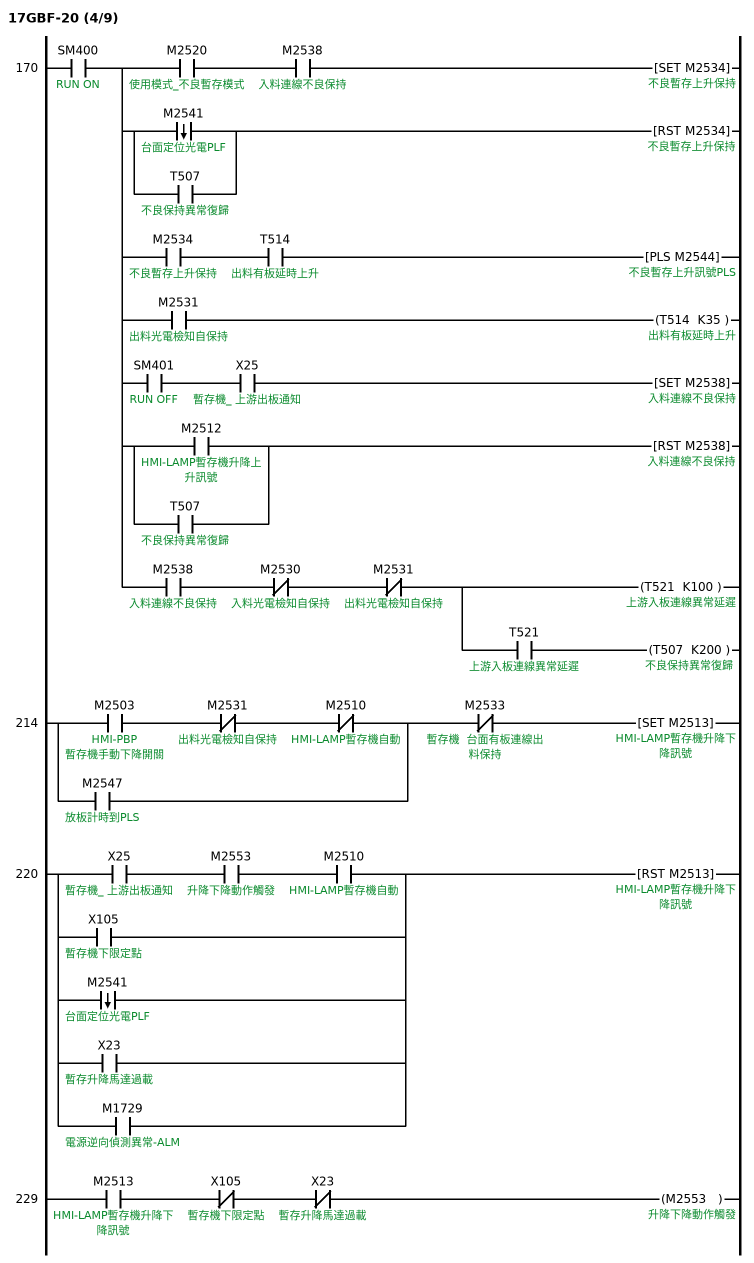
[picture p144: ladder of 17GBF-20, rungs at steps 170 to 229]
170   LD      SM400  ; RUN ON
      MPS
      AND     M2520  ; 使用模式_不良暫存模式
      AND     M2538  ; 入料連線不良保持
      SET     M2534  ; 不良暫存上升保持
      MRD
      LDF     M2541  ; 台面定位光電PLF
      OR      T507  ; 不良保持異常復歸
      ANB
      RST     M2534  ; 不良暫存上升保持
      MRD
      AND     M2534  ; 不良暫存上升保持
      AND     T514  ; 出料有板延時上升
      PLS     M2544  ; 不良暫存上升訊號PLS
      MRD
      AND     M2531  ; 出料光電檢知自保持
      OUT     T514 K35  ; 出料有板延時上升
      MRD
      AND     SM401  ; RUN OFF
      AND     X25  ; 暫存機_ 上游出板通知
      SET     M2538  ; 入料連線不良保持
      MRD
      LD      M2512  ; HMI-LAMP暫存機升降上升訊號
      OR      T507  ; 不良保持異常復歸
      ANB
      RST     M2538  ; 入料連線不良保持
      MPP
      AND     M2538  ; 入料連線不良保持
      ANI     M2530  ; 入料光電檢知自保持
      ANI     M2531  ; 出料光電檢知自保持
      OUT     T521 K100  ; 上游入板連線異常延遲
      AND     T521  ; 上游入板連線異常延遲
      OUT     T507 K200  ; 不良保持異常復歸
214   LD      M2503  ; HMI-PBP 暫存機手動下降開關
      ANI     M2531  ; 出料光電檢知自保持
      ANI     M2510  ; HMI-LAMP暫存機自動
      OR      M2547  ; 放板計時到PLS
      ANI     M2533  ; 暫存機  台面有板連線出料保持
      SET     M2513  ; HMI-LAMP暫存機升降下降訊號
220   LD      X25  ; 暫存機_ 上游出板通知
      AND     M2553  ; 升降下降動作觸發
      AND     M2510  ; HMI-LAMP暫存機自動
      OR      X105  ; 暫存機下限定點
      ORF     M2541  ; 台面定位光電PLF
      OR      X23  ; 暫存升降馬達過載
      OR      M1729  ; 電源逆向偵測異常-ALM
      RST     M2513  ; HMI-LAMP暫存機升降下降訊號
229   LD      M2513  ; HMI-LAMP暫存機升降下降訊號
      ANI     X105  ; 暫存機下限定點
      ANI     X23  ; 暫存升降馬達過載
      OUT     M2553  ; 升降下降動作觸發
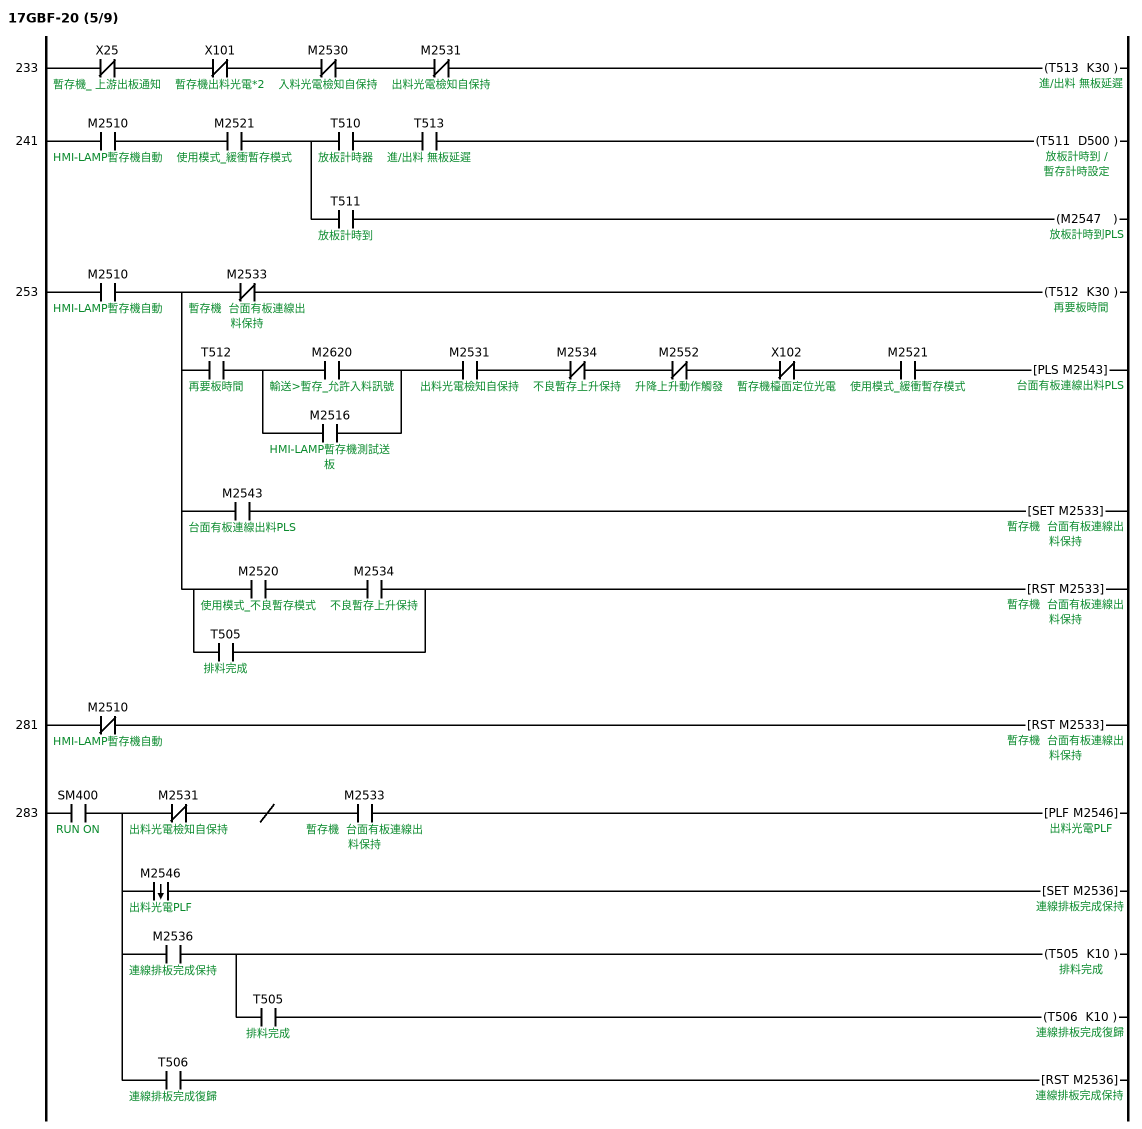
233   LDI     X25  ; 暫存機_ 上游出板通知
      ANI     X101  ; 暫存機出料光電*2
      ANI     M2530  ; 入料光電檢知自保持
      ANI     M2531  ; 出料光電檢知自保持
      OUT     T513 K30  ; 進/出料 無板延遲
241   LD      M2510  ; HMI-LAMP暫存機自動
      AND     M2521  ; 使用模式_緩衝暫存模式
      MPS
      AND     T510  ; 放板計時器
      AND     T513  ; 進/出料 無板延遲
      OUT     T511 D500  ; 放板計時到 / 暫存計時設定
      MPP
      AND     T511  ; 放板計時到
      OUT     M2547  ; 放板計時到PLS
253   LD      M2510  ; HMI-LAMP暫存機自動
      MPS
      ANI     M2533  ; 暫存機  台面有板連線出料保持
      OUT     T512 K30  ; 再要板時間
      MRD
      AND     T512  ; 再要板時間
      LD      M2620  ; 輸送>暫存_允許入料訊號
      OR      M2516  ; HMI-LAMP暫存機測試送板
      ANB
      AND     M2531  ; 出料光電檢知自保持
      ANI     M2534  ; 不良暫存上升保持
      ANI     M2552  ; 升降上升動作觸發
      ANI     X102  ; 暫存機檯面定位光電
      AND     M2521  ; 使用模式_緩衝暫存模式
      PLS     M2543  ; 台面有板連線出料PLS
      MRD
      AND     M2543  ; 台面有板連線出料PLS
      SET     M2533  ; 暫存機  台面有板連線出料保持
      MPP
      LD      M2520  ; 使用模式_不良暫存模式
      AND     M2534  ; 不良暫存上升保持
      OR      T505  ; 排料完成
      ANB
      RST     M2533  ; 暫存機  台面有板連線出料保持
281   LDI     M2510  ; HMI-LAMP暫存機自動
      RST     M2533  ; 暫存機  台面有板連線出料保持
283   LD      SM400  ; RUN ON
      MPS
      ANI     M2531  ; 出料光電檢知自保持
      INV
      AND     M2533  ; 暫存機  台面有板連線出料保持
      PLF     M2546  ; 出料光電PLF
      MRD
      ANDF    M2546  ; 出料光電PLF
      SET     M2536  ; 連線排板完成保持
      MRD
      AND     M2536  ; 連線排板完成保持
      OUT     T505 K10  ; 排料完成
      AND     T505  ; 排料完成
      OUT     T506 K10  ; 連線排板完成復歸
      MPP
      AND     T506  ; 連線排板完成復歸
      RST     M2536  ; 連線排板完成保持
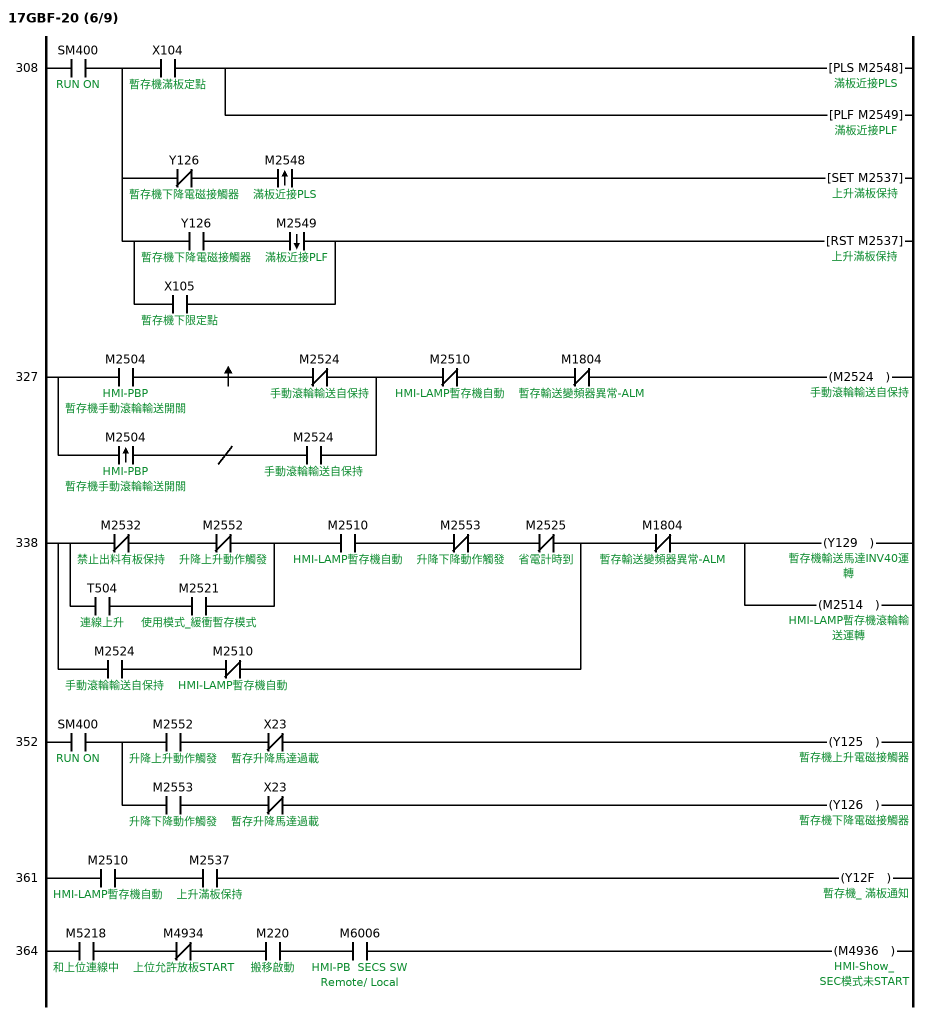
308   LD      SM400  ; RUN ON
      MPS
      AND     X104  ; 暫存機滿板定點
      PLS     M2548  ; 滿板近接PLS
      PLF     M2549  ; 滿板近接PLF
      MRD
      ANI     Y126  ; 暫存機下降電磁接觸器
      ANDP    M2548  ; 滿板近接PLS
      SET     M2537  ; 上升滿板保持
      MPP
      LD      Y126  ; 暫存機下降電磁接觸器
      ANDF    M2549  ; 滿板近接PLF
      OR      X105  ; 暫存機下限定點
      ANB
      RST     M2537  ; 上升滿板保持
327   LD      M2504  ; HMI-PBP 暫存機手動滾輪輸送開關
      MEP
      ANI     M2524  ; 手動滾輪輸送自保持
      LDP     M2504  ; HMI-PBP 暫存機手動滾輪輸送開關
      INV
      AND     M2524  ; 手動滾輪輸送自保持
      ORB
      ANI     M2510  ; HMI-LAMP暫存機自動
      ANI     M1804  ; 暫存輸送變頻器異常-ALM
      OUT     M2524  ; 手動滾輪輸送自保持
338   LDI     M2532  ; 禁止出料有板保持
      ANI     M2552  ; 升降上升動作觸發
      LD      T504  ; 連線上升
      AND     M2521  ; 使用模式_緩衝暫存模式
      ORB
      AND     M2510  ; HMI-LAMP暫存機自動
      ANI     M2553  ; 升降下降動作觸發
      ANI     M2525  ; 省電計時到
      LD      M2524  ; 手動滾輪輸送自保持
      ANI     M2510  ; HMI-LAMP暫存機自動
      ORB
      ANI     M1804  ; 暫存輸送變頻器異常-ALM
      OUT     Y129  ; 暫存機輸送馬達INV40運轉
      OUT     M2514  ; HMI-LAMP暫存機滾輪輸送運轉
352   LD      SM400  ; RUN ON
      MPS
      AND     M2552  ; 升降上升動作觸發
      ANI     X23  ; 暫存升降馬達過載
      OUT     Y125  ; 暫存機上升電磁接觸器
      MPP
      AND     M2553  ; 升降下降動作觸發
      ANI     X23  ; 暫存升降馬達過載
      OUT     Y126  ; 暫存機下降電磁接觸器
361   LD      M2510  ; HMI-LAMP暫存機自動
      AND     M2537  ; 上升滿板保持
      OUT     Y12F  ; 暫存機_ 滿板通知
364   LD      M5218  ; 和上位連線中
      ANI     M4934  ; 上位允許放板START
      AND     M220  ; 搬移啟動
      AND     M6006  ; HMI-PB  SECS SW  Remote/ Local
      OUT     M4936  ; HMI-Show_SEC模式未START
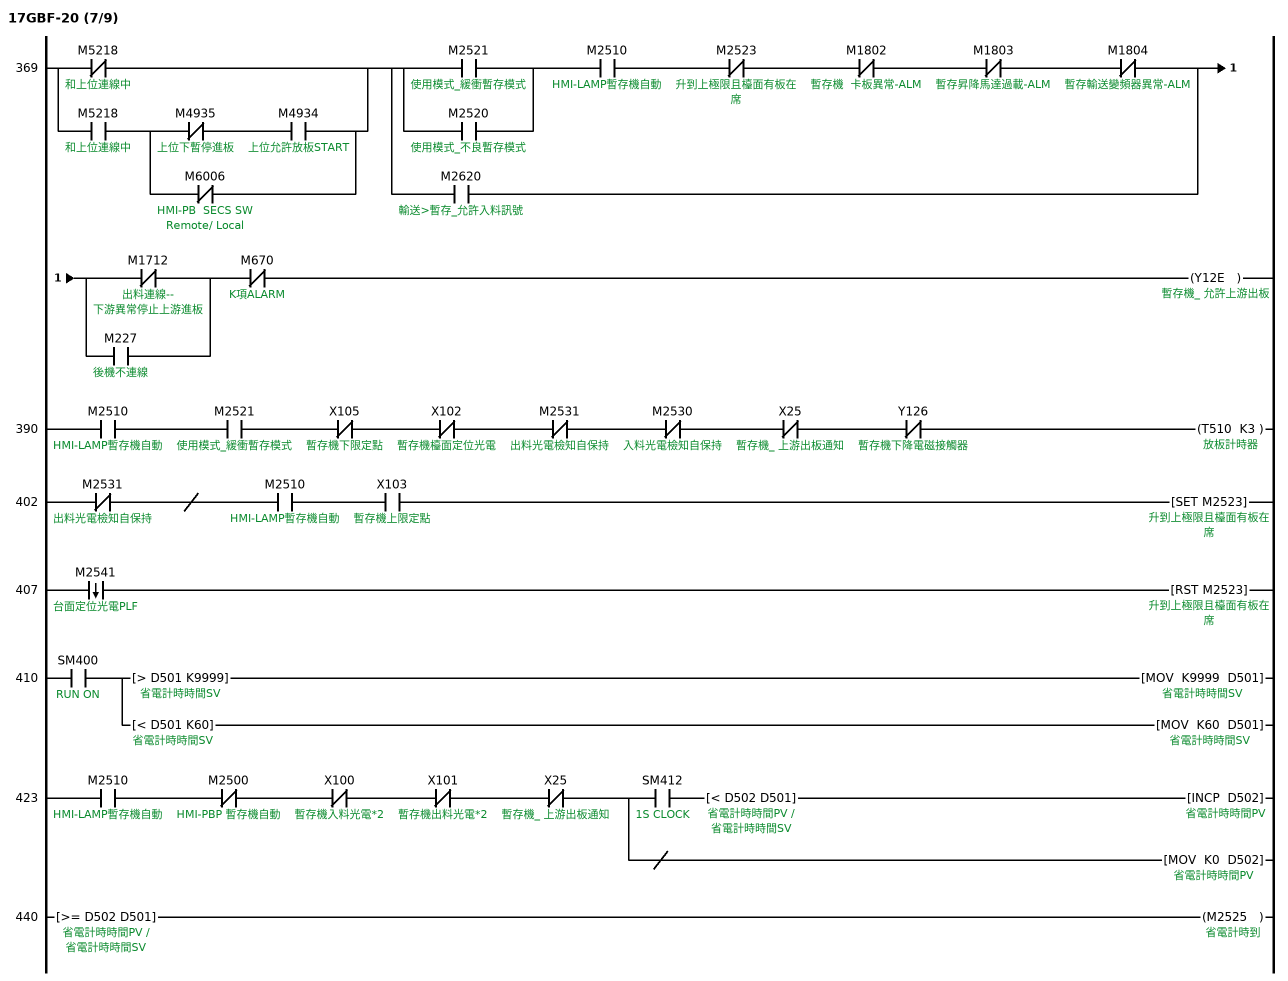
369   LDI     M5218  ; 和上位連線中
      LD      M5218  ; 和上位連線中
      LDI     M4935  ; 上位下暫停進板
      AND     M4934  ; 上位允許放板START
      ORI     M6006  ; HMI-PB  SECS SW  Remote/ Local
      ANB
      ORB
      LD      M2521  ; 使用模式_緩衝暫存模式
      OR      M2520  ; 使用模式_不良暫存模式
      AND     M2510  ; HMI-LAMP暫存機自動
      ANI     M2523  ; 升到上極限且檯面有板在席
      ANI     M1802  ; 暫存機  卡板異常-ALM
      ANI     M1803  ; 暫存昇降馬達過載-ALM
      ANI     M1804  ; 暫存輸送變頻器異常-ALM
      OR      M2620  ; 輸送>暫存_允許入料訊號
      ANB
      LDI     M1712  ; 出料連線--下游異常停止上游進板
      OR      M227  ; 後機不連線
      ANB
      ANI     M670  ; K項ALARM
      OUT     Y12E  ; 暫存機_ 允許上游出板
390   LD      M2510  ; HMI-LAMP暫存機自動
      AND     M2521  ; 使用模式_緩衝暫存模式
      ANI     X105  ; 暫存機下限定點
      ANI     X102  ; 暫存機檯面定位光電
      ANI     M2531  ; 出料光電檢知自保持
      ANI     M2530  ; 入料光電檢知自保持
      ANI     X25  ; 暫存機_ 上游出板通知
      ANI     Y126  ; 暫存機下降電磁接觸器
      OUT     T510 K3  ; 放板計時器
402   LDI     M2531  ; 出料光電檢知自保持
      INV
      AND     M2510  ; HMI-LAMP暫存機自動
      AND     X103  ; 暫存機上限定點
      SET     M2523  ; 升到上極限且檯面有板在席
407   LDF     M2541  ; 台面定位光電PLF
      RST     M2523  ; 升到上極限且檯面有板在席
410   LD      SM400  ; RUN ON
      MPS
      AND>    D501 K9999  ; 省電計時時間SV
      MOV     K9999 D501
      MPP
      AND<    D501 K60  ; 省電計時時間SV
      MOV     K60 D501
423   LD      M2510  ; HMI-LAMP暫存機自動
      ANI     M2500  ; HMI-PBP 暫存機自動
      ANI     X100  ; 暫存機入料光電*2
      ANI     X101  ; 暫存機出料光電*2
      ANI     X25  ; 暫存機_ 上游出板通知
      MPS
      AND     SM412  ; 1S CLOCK
      AND<    D502 D501  ; 省電計時時間PV / 省電計時時間SV
      INCP    D502
      MPP
      INV
      MOV     K0 D502
440   LD>=    D502 D501  ; 省電計時時間PV / 省電計時時間SV
      OUT     M2525  ; 省電計時到
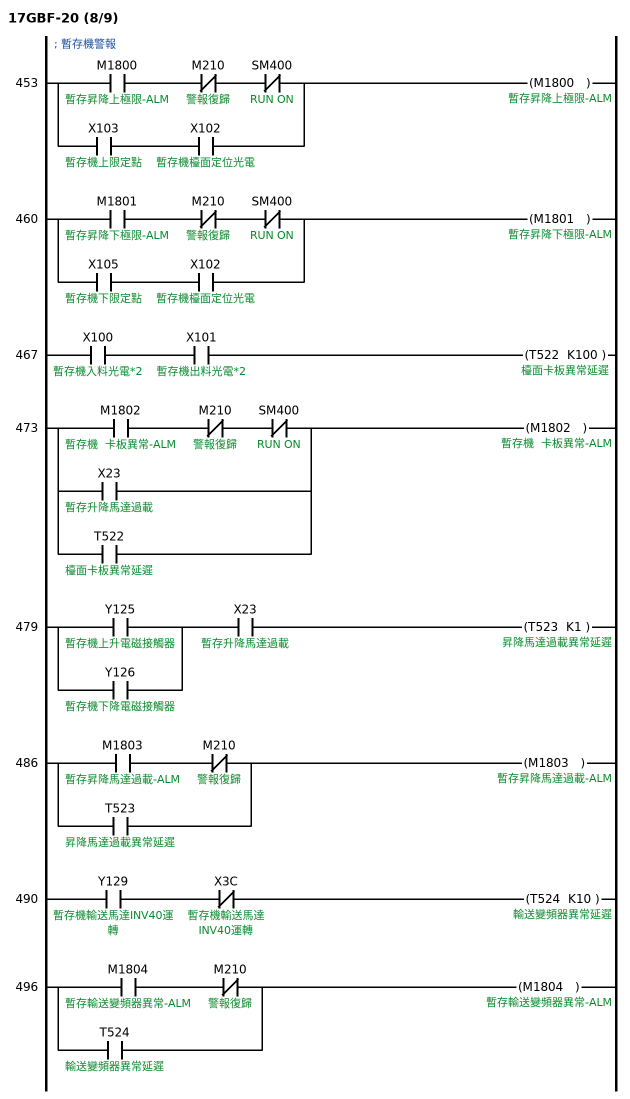
; 暫存機警報
453   LD      M1800  ; 暫存昇降上極限-ALM
      ANI     M210  ; 警報復歸
      ANI     SM400  ; RUN ON
      LD      X103  ; 暫存機上限定點
      AND     X102  ; 暫存機檯面定位光電
      ORB
      OUT     M1800  ; 暫存昇降上極限-ALM
460   LD      M1801  ; 暫存昇降下極限-ALM
      ANI     M210  ; 警報復歸
      ANI     SM400  ; RUN ON
      LD      X105  ; 暫存機下限定點
      AND     X102  ; 暫存機檯面定位光電
      ORB
      OUT     M1801  ; 暫存昇降下極限-ALM
467   LD      X100  ; 暫存機入料光電*2
      AND     X101  ; 暫存機出料光電*2
      OUT     T522 K100  ; 檯面卡板異常延遲
473   LD      M1802  ; 暫存機  卡板異常-ALM
      ANI     M210  ; 警報復歸
      ANI     SM400  ; RUN ON
      OR      X23  ; 暫存升降馬達過載
      OR      T522  ; 檯面卡板異常延遲
      OUT     M1802  ; 暫存機  卡板異常-ALM
479   LD      Y125  ; 暫存機上升電磁接觸器
      OR      Y126  ; 暫存機下降電磁接觸器
      AND     X23  ; 暫存升降馬達過載
      OUT     T523 K1  ; 昇降馬達過載異常延遲
486   LD      M1803  ; 暫存昇降馬達過載-ALM
      ANI     M210  ; 警報復歸
      OR      T523  ; 昇降馬達過載異常延遲
      OUT     M1803  ; 暫存昇降馬達過載-ALM
490   LD      Y129  ; 暫存機輸送馬達INV40運轉
      ANI     X3C  ; 暫存機輸送馬達  INV40運轉
      OUT     T524 K10  ; 輸送變頻器異常延遲
496   LD      M1804  ; 暫存輸送變頻器異常-ALM
      ANI     M210  ; 警報復歸
      OR      T524  ; 輸送變頻器異常延遲
      OUT     M1804  ; 暫存輸送變頻器異常-ALM
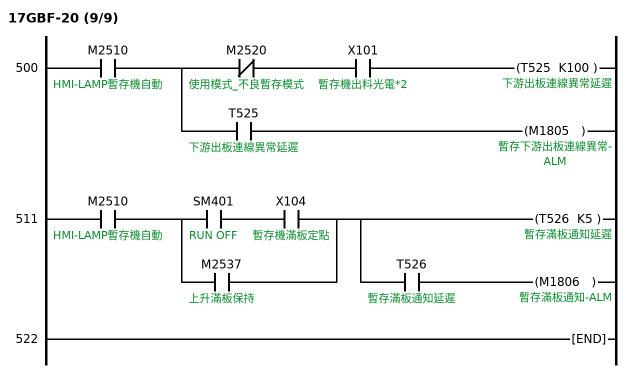
500   LD      M2510  ; HMI-LAMP暫存機自動
      MPS
      ANI     M2520  ; 使用模式_不良暫存模式
      AND     X101  ; 暫存機出料光電*2
      OUT     T525 K100  ; 下游出板連線異常延遲
      MPP
      AND     T525  ; 下游出板連線異常延遲
      OUT     M1805  ; 暫存下游出板連線異常-ALM
511   LD      M2510  ; HMI-LAMP暫存機自動
      LD      SM401  ; RUN OFF
      AND     X104  ; 暫存機滿板定點
      OR      M2537  ; 上升滿板保持
      ANB
      OUT     T526 K5  ; 暫存滿板通知延遲
      AND     T526  ; 暫存滿板通知延遲
      OUT     M1806  ; 暫存滿板通知-ALM
522   END
END_PROGRAM

PROGRAM 18GCV
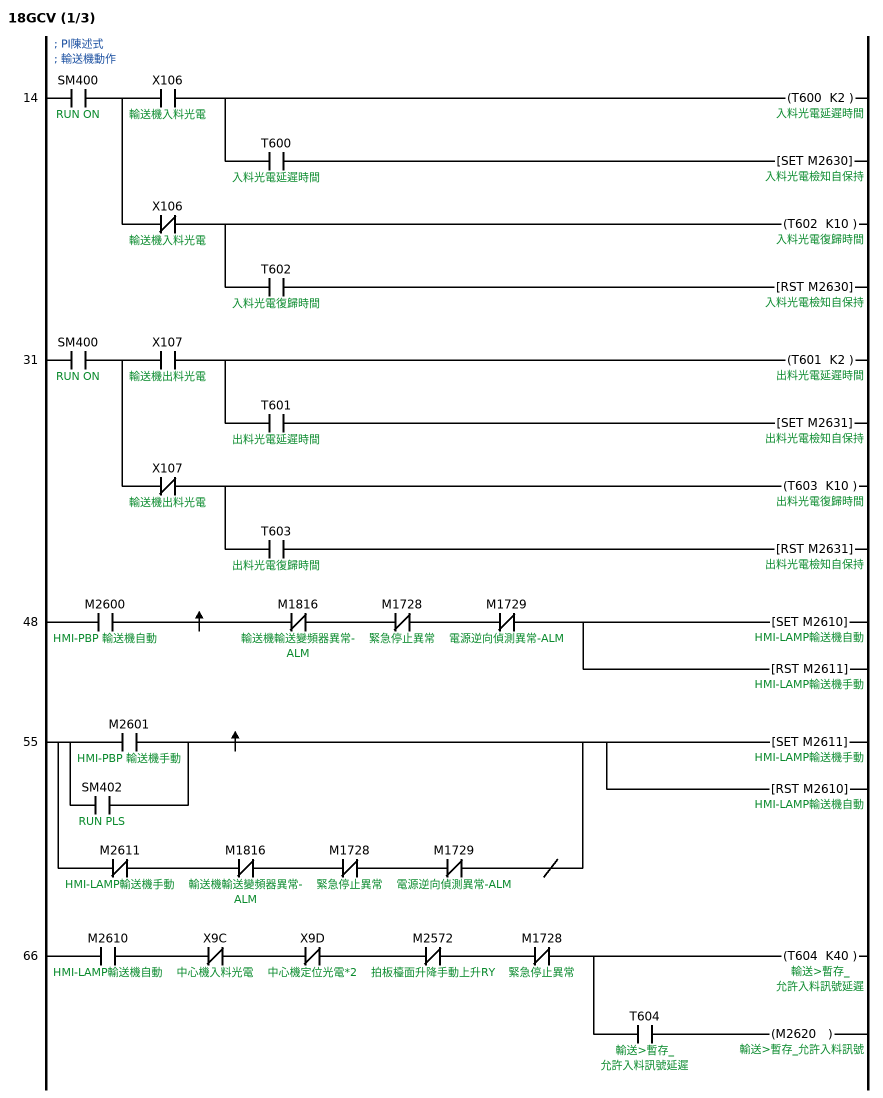
; PI陳述式
; 輸送機動作
14    LD      SM400  ; RUN ON
      MPS
      AND     X106  ; 輸送機入料光電
      OUT     T600 K2  ; 入料光電延遲時間
      AND     T600  ; 入料光電延遲時間
      SET     M2630  ; 入料光電檢知自保持
      MPP
      ANI     X106  ; 輸送機入料光電
      OUT     T602 K10  ; 入料光電復歸時間
      AND     T602  ; 入料光電復歸時間
      RST     M2630  ; 入料光電檢知自保持
31    LD      SM400  ; RUN ON
      MPS
      AND     X107  ; 輸送機出料光電
      OUT     T601 K2  ; 出料光電延遲時間
      AND     T601  ; 出料光電延遲時間
      SET     M2631  ; 出料光電檢知自保持
      MPP
      ANI     X107  ; 輸送機出料光電
      OUT     T603 K10  ; 出料光電復歸時間
      AND     T603  ; 出料光電復歸時間
      RST     M2631  ; 出料光電檢知自保持
48    LD      M2600  ; HMI-PBP 輸送機自動
      MEP
      ANI     M1816  ; 輸送機輸送變頻器異常-ALM
      ANI     M1728  ; 緊急停止異常
      ANI     M1729  ; 電源逆向偵測異常-ALM
      SET     M2610  ; HMI-LAMP輸送機自動
      RST     M2611  ; HMI-LAMP輸送機手動
55    LD      M2601  ; HMI-PBP 輸送機手動
      OR      SM402  ; RUN PLS
      MEP
      LDI     M2611  ; HMI-LAMP輸送機手動
      ANI     M1816  ; 輸送機輸送變頻器異常-ALM
      ANI     M1728  ; 緊急停止異常
      ANI     M1729  ; 電源逆向偵測異常-ALM
      INV
      ORB
      SET     M2611  ; HMI-LAMP輸送機手動
      RST     M2610  ; HMI-LAMP輸送機自動
66    LD      M2610  ; HMI-LAMP輸送機自動
      ANI     X9C  ; 中心機入料光電
      ANI     X9D  ; 中心機定位光電*2
      ANI     M2572  ; 拍板檯面升降手動上升RY
      ANI     M1728  ; 緊急停止異常
      OUT     T604 K40  ; 輸送>暫存_允許入料訊號延遲
      AND     T604  ; 輸送>暫存_允許入料訊號延遲
      OUT     M2620  ; 輸送>暫存_允許入料訊號
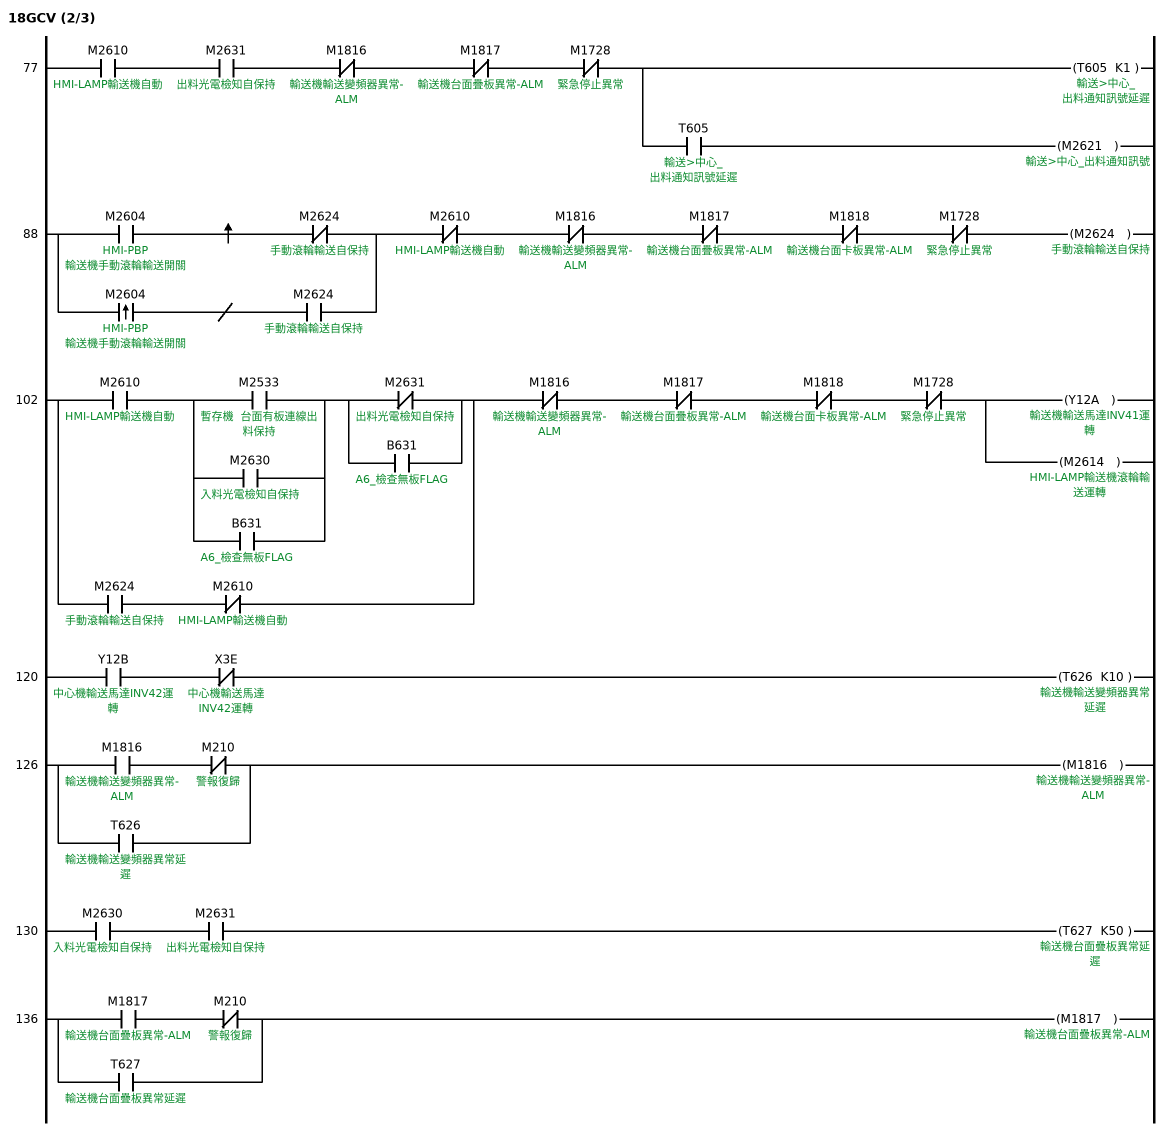
77    LD      M2610  ; HMI-LAMP輸送機自動
      AND     M2631  ; 出料光電檢知自保持
      ANI     M1816  ; 輸送機輸送變頻器異常-ALM
      ANI     M1817  ; 輸送機台面疊板異常-ALM
      ANI     M1728  ; 緊急停止異常
      OUT     T605 K1  ; 輸送>中心_出料通知訊號延遲
      AND     T605  ; 輸送>中心_出料通知訊號延遲
      OUT     M2621  ; 輸送>中心_出料通知訊號
88    LD      M2604  ; HMI-PBP 輸送機手動滾輪輸送開關
      MEP
      ANI     M2624  ; 手動滾輪輸送自保持
      LDP     M2604  ; HMI-PBP 輸送機手動滾輪輸送開關
      INV
      AND     M2624  ; 手動滾輪輸送自保持
      ORB
      ANI     M2610  ; HMI-LAMP輸送機自動
      ANI     M1816  ; 輸送機輸送變頻器異常-ALM
      ANI     M1817  ; 輸送機台面疊板異常-ALM
      ANI     M1818  ; 輸送機台面卡板異常-ALM
      ANI     M1728  ; 緊急停止異常
      OUT     M2624  ; 手動滾輪輸送自保持
102   LD      M2610  ; HMI-LAMP輸送機自動
      LD      M2533  ; 暫存機  台面有板連線出料保持
      OR      M2630  ; 入料光電檢知自保持
      OR      B631  ; A6_檢查無板FLAG
      ANB
      LDI     M2631  ; 出料光電檢知自保持
      OR      B631  ; A6_檢查無板FLAG
      ANB
      LD      M2624  ; 手動滾輪輸送自保持
      ANI     M2610  ; HMI-LAMP輸送機自動
      ORB
      ANI     M1816  ; 輸送機輸送變頻器異常-ALM
      ANI     M1817  ; 輸送機台面疊板異常-ALM
      ANI     M1818  ; 輸送機台面卡板異常-ALM
      ANI     M1728  ; 緊急停止異常
      OUT     Y12A  ; 輸送機輸送馬達INV41運轉
      OUT     M2614  ; HMI-LAMP輸送機滾輪輸送運轉
120   LD      Y12B  ; 中心機輸送馬達INV42運轉
      ANI     X3E  ; 中心機輸送馬達  INV42運轉
      OUT     T626 K10  ; 輸送機輸送變頻器異常延遲
126   LD      M1816  ; 輸送機輸送變頻器異常-ALM
      ANI     M210  ; 警報復歸
      OR      T626  ; 輸送機輸送變頻器異常延遲
      OUT     M1816  ; 輸送機輸送變頻器異常-ALM
130   LD      M2630  ; 入料光電檢知自保持
      AND     M2631  ; 出料光電檢知自保持
      OUT     T627 K50  ; 輸送機台面疊板異常延遲
136   LD      M1817  ; 輸送機台面疊板異常-ALM
      ANI     M210  ; 警報復歸
      OR      T627  ; 輸送機台面疊板異常延遲
      OUT     M1817  ; 輸送機台面疊板異常-ALM
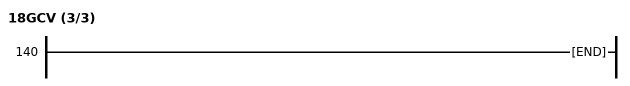
140   END
END_PROGRAM

PROGRAM 19GTC-7
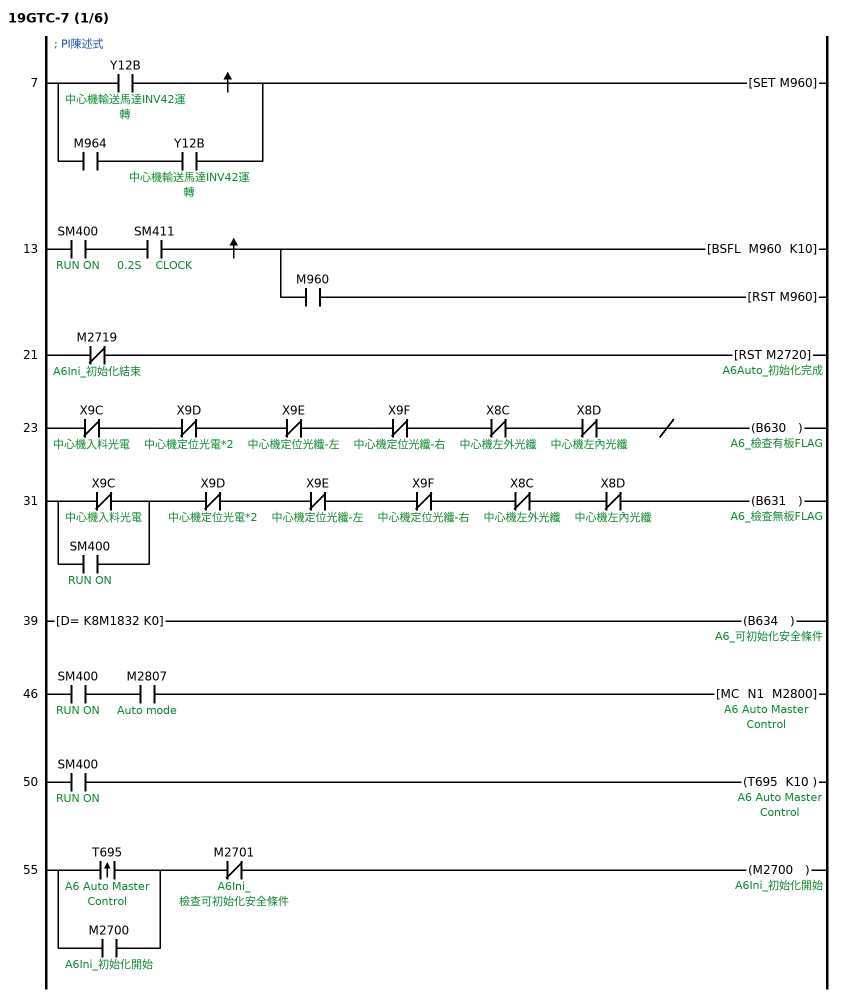
; PI陳述式
7     LD      Y12B  ; 中心機輸送馬達INV42運轉
      MEP
      LD      M964
      AND     Y12B  ; 中心機輸送馬達INV42運轉
      ORB
      SET     M960
13    LD      SM400  ; RUN ON
      AND     SM411  ; 0.2S    CLOCK
      MEP
      BSFL    M960 K10
      AND     M960
      RST     M960
21    LDI     M2719  ; A6Ini_初始化結束
      RST     M2720  ; A6Auto_初始化完成
23    LDI     X9C  ; 中心機入料光電
      ANI     X9D  ; 中心機定位光電*2
      ANI     X9E  ; 中心機定位光纖-左
      ANI     X9F  ; 中心機定位光纖-右
      ANI     X8C  ; 中心機左外光纖
      ANI     X8D  ; 中心機左內光纖
      INV
      OUT     B630  ; A6_檢查有板FLAG
31    LDI     X9C  ; 中心機入料光電
      OR      SM400  ; RUN ON
      ANI     X9D  ; 中心機定位光電*2
      ANI     X9E  ; 中心機定位光纖-左
      ANI     X9F  ; 中心機定位光纖-右
      ANI     X8C  ; 中心機左外光纖
      ANI     X8D  ; 中心機左內光纖
      OUT     B631  ; A6_檢查無板FLAG
39    LDD=    K8M1832 K0
      OUT     B634  ; A6_可初始化安全條件
46    LD      SM400  ; RUN ON
      AND     M2807  ; Auto mode
      MC      N1 M2800  ; A6 Auto Master Control
50    LD      SM400  ; RUN ON
      OUT     T695 K10  ; A6 Auto Master Control
55    LDP     T695  ; A6 Auto Master Control
      OR      M2700  ; A6Ini_初始化開始
      ANI     M2701  ; A6Ini_檢查可初始化安全條件
      OUT     M2700  ; A6Ini_初始化開始
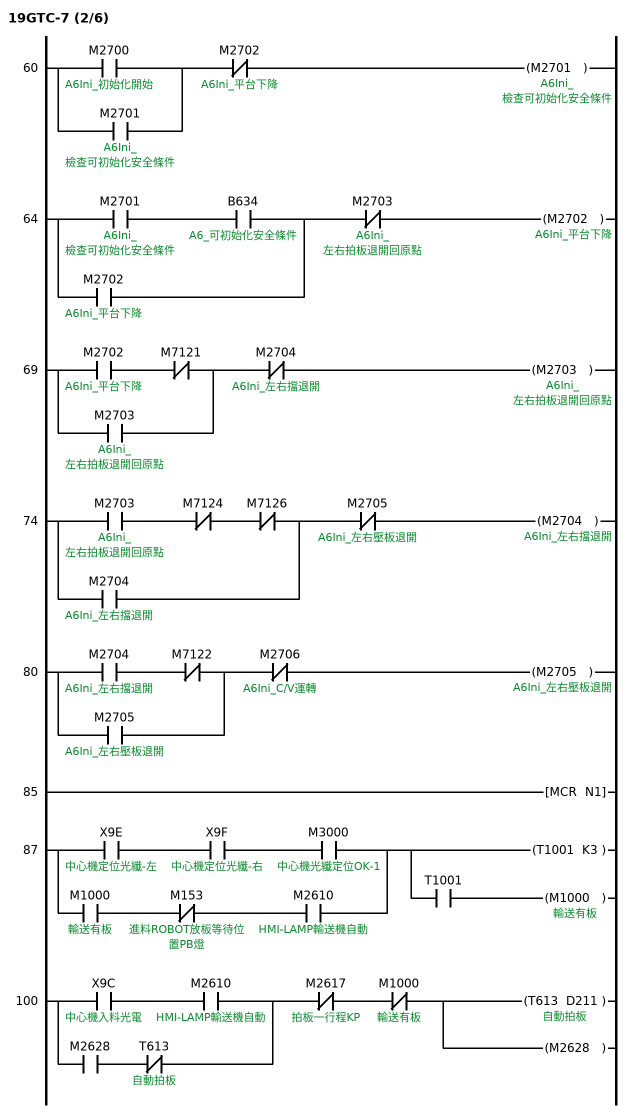
60    LD      M2700  ; A6Ini_初始化開始
      OR      M2701  ; A6Ini_檢查可初始化安全條件
      ANI     M2702  ; A6Ini_平台下降
      OUT     M2701  ; A6Ini_檢查可初始化安全條件
64    LD      M2701  ; A6Ini_檢查可初始化安全條件
      AND     B634  ; A6_可初始化安全條件
      OR      M2702  ; A6Ini_平台下降
      ANI     M2703  ; A6Ini_左右拍板退開回原點
      OUT     M2702  ; A6Ini_平台下降
69    LD      M2702  ; A6Ini_平台下降
      ANI     M7121
      OR      M2703  ; A6Ini_左右拍板退開回原點
      ANI     M2704  ; A6Ini_左右擋退開
      OUT     M2703  ; A6Ini_左右拍板退開回原點
74    LD      M2703  ; A6Ini_左右拍板退開回原點
      ANI     M7124
      ANI     M7126
      OR      M2704  ; A6Ini_左右擋退開
      ANI     M2705  ; A6Ini_左右壓板退開
      OUT     M2704  ; A6Ini_左右擋退開
80    LD      M2704  ; A6Ini_左右擋退開
      ANI     M7122
      OR      M2705  ; A6Ini_左右壓板退開
      ANI     M2706  ; A6Ini_C/V運轉
      OUT     M2705  ; A6Ini_左右壓板退開
85    MCR     N1
87    LD      X9E  ; 中心機定位光纖-左
      AND     X9F  ; 中心機定位光纖-右
      AND     M3000  ; 中心機光纖定位OK-1
      LD      M1000  ; 輸送有板
      ANI     M153  ; 進料ROBOT放板等待位置PB燈
      AND     M2610  ; HMI-LAMP輸送機自動
      ORB
      OUT     T1001 K3
      AND     T1001
      OUT     M1000  ; 輸送有板
100   LD      X9C  ; 中心機入料光電
      AND     M2610  ; HMI-LAMP輸送機自動
      LD      M2628
      ANI     T613  ; 自動拍板
      ORB
      ANI     M2617  ; 拍板一行程KP
      ANI     M1000  ; 輸送有板
      OUT     T613 D211  ; 自動拍板
      OUT     M2628
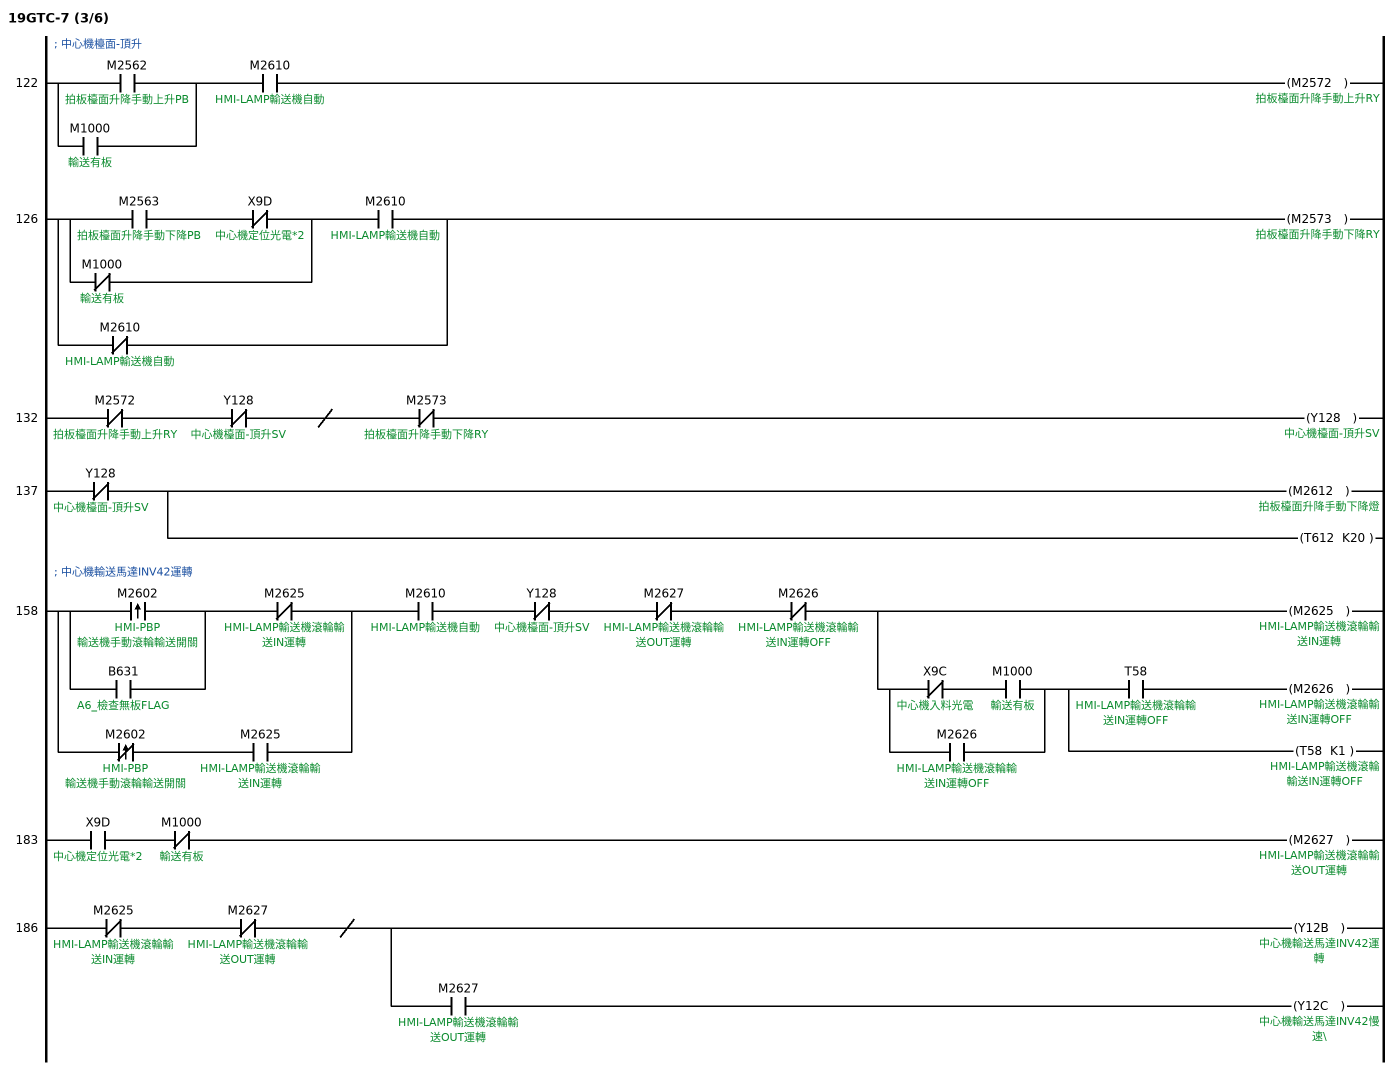
; 中心機檯面-頂升
122   LD      M2562  ; 拍板檯面升降手動上升PB
      OR      M1000  ; 輸送有板
      AND     M2610  ; HMI-LAMP輸送機自動
      OUT     M2572  ; 拍板檯面升降手動上升RY
126   LD      M2563  ; 拍板檯面升降手動下降PB
      ANI     X9D  ; 中心機定位光電*2
      ORI     M1000  ; 輸送有板
      AND     M2610  ; HMI-LAMP輸送機自動
      ORI     M2610  ; HMI-LAMP輸送機自動
      OUT     M2573  ; 拍板檯面升降手動下降RY
132   LDI     M2572  ; 拍板檯面升降手動上升RY
      ANI     Y128  ; 中心機檯面-頂升SV
      INV
      ANI     M2573  ; 拍板檯面升降手動下降RY
      OUT     Y128  ; 中心機檯面-頂升SV
137   LDI     Y128  ; 中心機檯面-頂升SV
      OUT     M2612  ; 拍板檯面升降手動下降燈
      OUT     T612 K20
; 中心機輸送馬達INV42運轉
158   LDP     M2602  ; HMI-PBP 輸送機手動滾輪輸送開關
      OR      B631  ; A6_檢查無板FLAG
      ANI     M2625  ; HMI-LAMP輸送機滾輪輸送IN運轉
      LDPI    M2602  ; HMI-PBP 輸送機手動滾輪輸送開關
      AND     M2625  ; HMI-LAMP輸送機滾輪輸送IN運轉
      ORB
      AND     M2610  ; HMI-LAMP輸送機自動
      ANI     Y128  ; 中心機檯面-頂升SV
      ANI     M2627  ; HMI-LAMP輸送機滾輪輸送OUT運轉
      ANI     M2626  ; HMI-LAMP輸送機滾輪輸送IN運轉OFF
      OUT     M2625  ; HMI-LAMP輸送機滾輪輸送IN運轉
      LDI     X9C  ; 中心機入料光電
      AND     M1000  ; 輸送有板
      OR      M2626  ; HMI-LAMP輸送機滾輪輸送IN運轉OFF
      ANB
      MPS
      AND     T58  ; HMI-LAMP輸送機滾輪輸送IN運轉OFF
      OUT     M2626  ; HMI-LAMP輸送機滾輪輸送IN運轉OFF
      MPP
      OUT     T58 K1  ; HMI-LAMP輸送機滾輪輸送IN運轉OFF
183   LD      X9D  ; 中心機定位光電*2
      ANI     M1000  ; 輸送有板
      OUT     M2627  ; HMI-LAMP輸送機滾輪輸送OUT運轉
186   LDI     M2625  ; HMI-LAMP輸送機滾輪輸送IN運轉
      ANI     M2627  ; HMI-LAMP輸送機滾輪輸送OUT運轉
      INV
      OUT     Y12B  ; 中心機輸送馬達INV42運轉
      AND     M2627  ; HMI-LAMP輸送機滾輪輸送OUT運轉
      OUT     Y12C  ; 中心機輸送馬達INV42慢速\
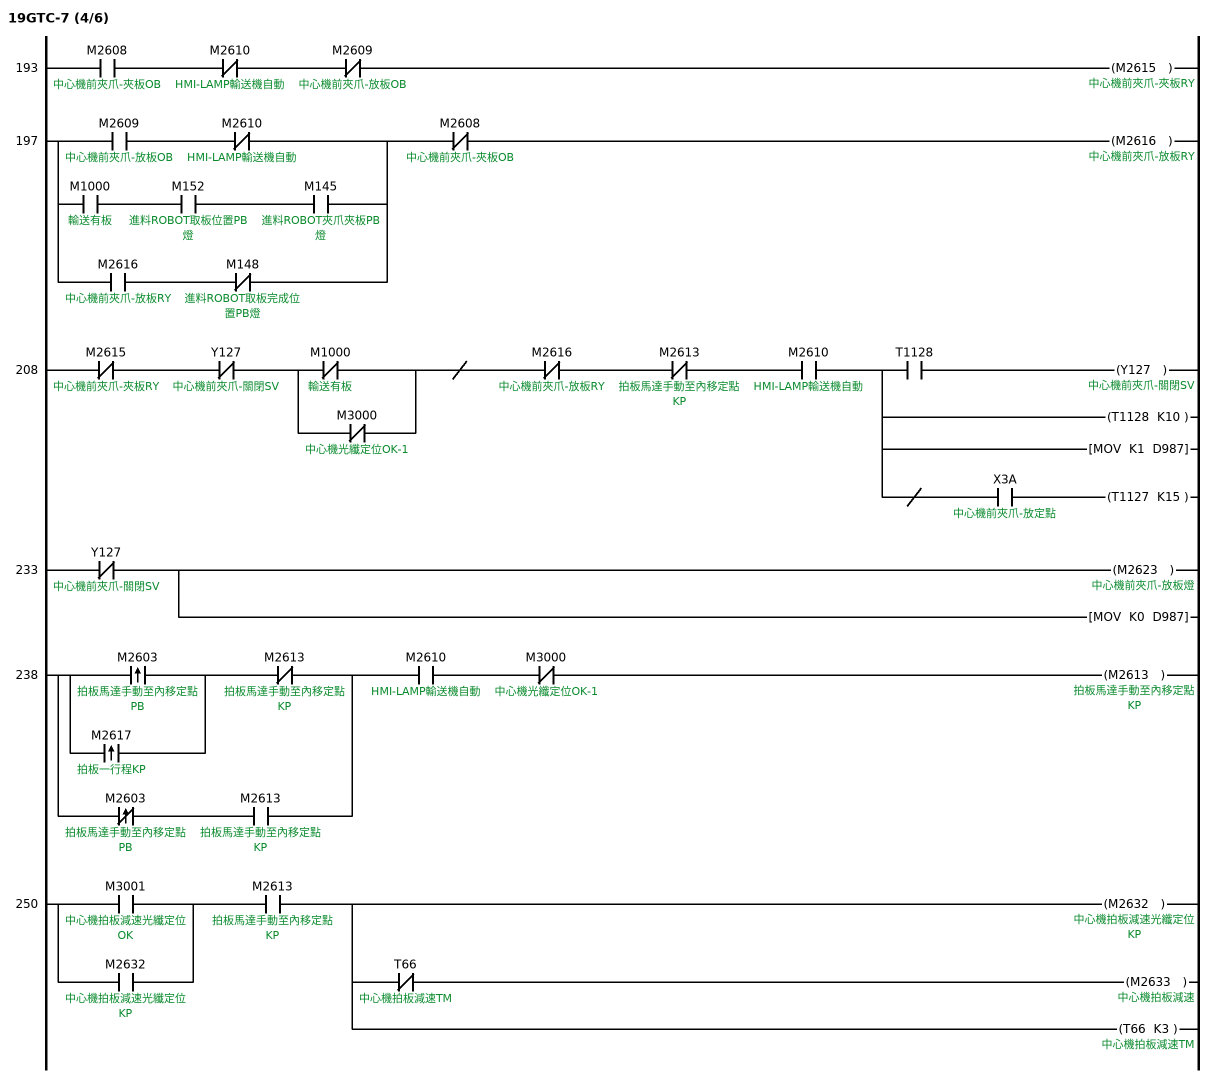
193   LD      M2608  ; 中心機前夾爪-夾板OB
      ANI     M2610  ; HMI-LAMP輸送機自動
      ANI     M2609  ; 中心機前夾爪-放板OB
      OUT     M2615  ; 中心機前夾爪-夾板RY
197   LD      M2609  ; 中心機前夾爪-放板OB
      ANI     M2610  ; HMI-LAMP輸送機自動
      LD      M1000  ; 輸送有板
      AND     M152  ; 進料ROBOT取板位置PB燈
      AND     M145  ; 進料ROBOT夾爪夾板PB燈
      ORB
      LD      M2616  ; 中心機前夾爪-放板RY
      ANI     M148  ; 進料ROBOT取板完成位置PB燈
      ORB
      ANI     M2608  ; 中心機前夾爪-夾板OB
      OUT     M2616  ; 中心機前夾爪-放板RY
208   LDI     M2615  ; 中心機前夾爪-夾板RY
      ANI     Y127  ; 中心機前夾爪-關閉SV
      LDI     M1000  ; 輸送有板
      ORI     M3000  ; 中心機光纖定位OK-1
      ANB
      INV
      ANI     M2616  ; 中心機前夾爪-放板RY
      ANI     M2613  ; 拍板馬達手動至內移定點KP
      AND     M2610  ; HMI-LAMP輸送機自動
      MPS
      AND     T1128
      OUT     Y127  ; 中心機前夾爪-關閉SV
      MPP
      OUT     T1128 K10
      MOV     K1 D987
      INV
      AND     X3A  ; 中心機前夾爪-放定點
      OUT     T1127 K15
233   LDI     Y127  ; 中心機前夾爪-關閉SV
      OUT     M2623  ; 中心機前夾爪-放板燈
      MOV     K0 D987
238   LDP     M2603  ; 拍板馬達手動至內移定點PB
      ORP     M2617  ; 拍板一行程KP
      ANI     M2613  ; 拍板馬達手動至內移定點KP
      LDPI    M2603  ; 拍板馬達手動至內移定點PB
      AND     M2613  ; 拍板馬達手動至內移定點KP
      ORB
      AND     M2610  ; HMI-LAMP輸送機自動
      ANI     M3000  ; 中心機光纖定位OK-1
      OUT     M2613  ; 拍板馬達手動至內移定點KP
250   LD      M3001  ; 中心機拍板減速光纖定位OK
      OR      M2632  ; 中心機拍板減速光纖定位KP
      AND     M2613  ; 拍板馬達手動至內移定點KP
      OUT     M2632  ; 中心機拍板減速光纖定位KP
      MPS
      ANI     T66  ; 中心機拍板減速TM
      OUT     M2633  ; 中心機拍板減速
      MPP
      OUT     T66 K3  ; 中心機拍板減速TM
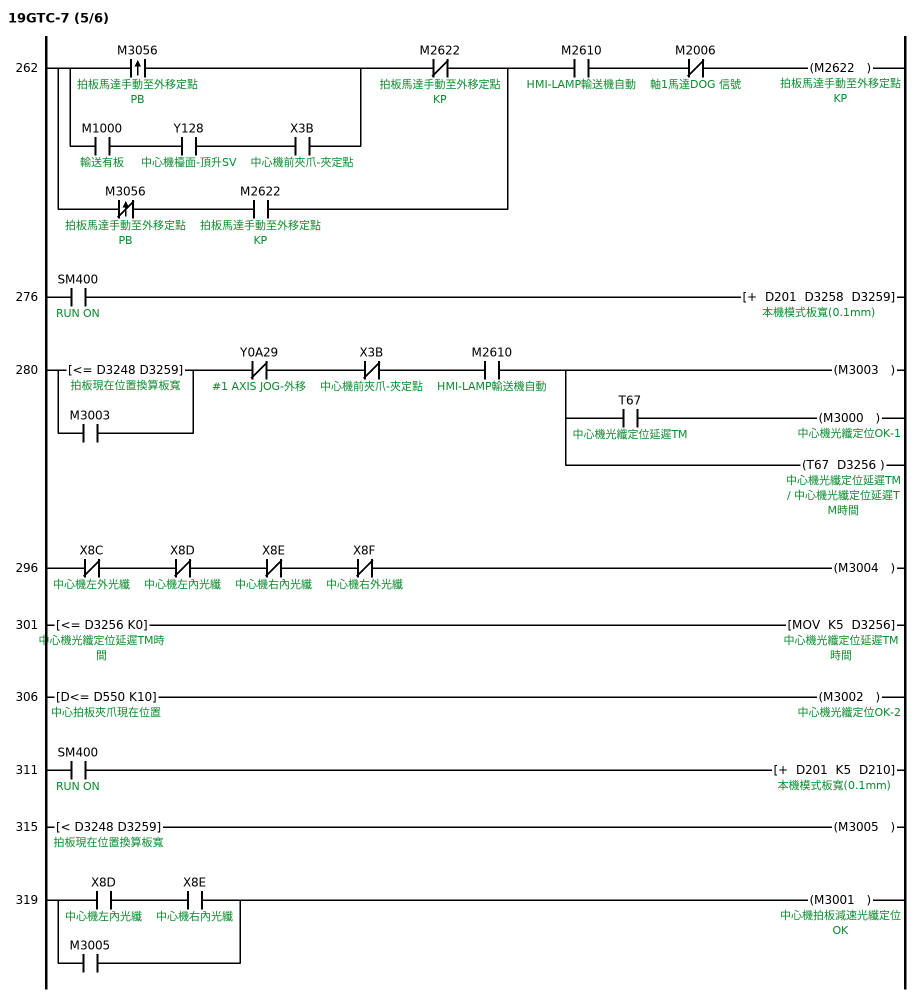
262   LDP     M3056  ; 拍板馬達手動至外移定點PB
      LD      M1000  ; 輸送有板
      AND     Y128  ; 中心機檯面-頂升SV
      AND     X3B  ; 中心機前夾爪-夾定點
      ORB
      ANI     M2622  ; 拍板馬達手動至外移定點KP
      LDPI    M3056  ; 拍板馬達手動至外移定點PB
      AND     M2622  ; 拍板馬達手動至外移定點KP
      ORB
      AND     M2610  ; HMI-LAMP輸送機自動
      ANI     M2006  ; 軸1馬達DOG 信號
      OUT     M2622  ; 拍板馬達手動至外移定點KP
276   LD      SM400  ; RUN ON
      +       D201 D3258 D3259  ; 本機模式板寬(0.1mm)
280   LD<=    D3248 D3259  ; 拍板現在位置換算板寬
      OR      M3003
      ANI     Y0A29  ; #1 AXIS JOG-外移
      ANI     X3B  ; 中心機前夾爪-夾定點
      AND     M2610  ; HMI-LAMP輸送機自動
      OUT     M3003
      MPS
      AND     T67  ; 中心機光纖定位延遲TM
      OUT     M3000  ; 中心機光纖定位OK-1
      MPP
      OUT     T67 D3256  ; 中心機光纖定位延遲TM / 中心機光纖定位延遲TM時間
296   LDI     X8C  ; 中心機左外光纖
      ANI     X8D  ; 中心機左內光纖
      ANI     X8E  ; 中心機右內光纖
      ANI     X8F  ; 中心機右外光纖
      OUT     M3004
301   LD<=    D3256 K0  ; 中心機光纖定位延遲TM時間
      MOV     K5 D3256
306   LDD<=   D550 K10  ; 中心拍板夾爪現在位置
      OUT     M3002  ; 中心機光纖定位OK-2
311   LD      SM400  ; RUN ON
      +       D201 K5 D210
315   LD<     D3248 D3259  ; 拍板現在位置換算板寬
      OUT     M3005
319   LD      X8D  ; 中心機左內光纖
      AND     X8E  ; 中心機右內光纖
      OR      M3005
      OUT     M3001  ; 中心機拍板減速光纖定位OK
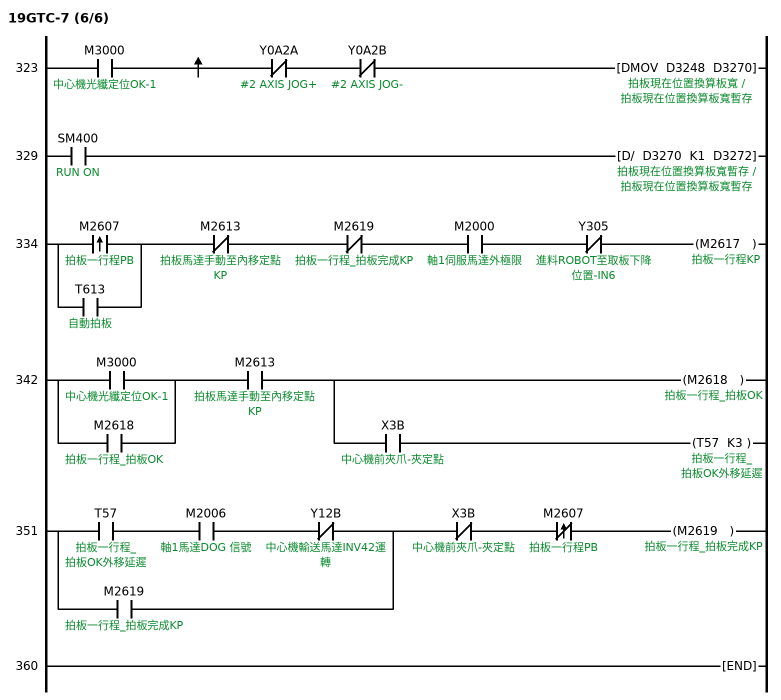
323   LD      M3000  ; 中心機光纖定位OK-1
      MEP
      ANI     Y0A2A  ; #2 AXIS JOG+
      ANI     Y0A2B  ; #2 AXIS JOG-
      DMOV    D3248 D3270  ; 拍板現在位置換算板寬暫存
329   LD      SM400  ; RUN ON
      D/      D3270 K1 D3272  ; 拍板現在位置換算板寬暫存
334   LDP     M2607  ; 拍板一行程PB
      OR      T613  ; 自動拍板
      ANI     M2613  ; 拍板馬達手動至內移定點KP
      ANI     M2619  ; 拍板一行程_拍板完成KP
      AND     M2000  ; 軸1伺服馬達外極限
      ANI     Y305  ; 進料ROBOT至取板下降位置-IN6
      OUT     M2617  ; 拍板一行程KP
342   LD      M3000  ; 中心機光纖定位OK-1
      OR      M2618  ; 拍板一行程_拍板OK
      AND     M2613  ; 拍板馬達手動至內移定點KP
      OUT     M2618  ; 拍板一行程_拍板OK
      AND     X3B  ; 中心機前夾爪-夾定點
      OUT     T57 K3  ; 拍板一行程_拍板OK外移延遲
351   LD      T57  ; 拍板一行程_拍板OK外移延遲
      AND     M2006  ; 軸1馬達DOG 信號
      ANI     Y12B  ; 中心機輸送馬達INV42運轉
      OR      M2619  ; 拍板一行程_拍板完成KP
      ANI     X3B  ; 中心機前夾爪-夾定點
      ANDPI   M2607  ; 拍板一行程PB
      OUT     M2619  ; 拍板一行程_拍板完成KP
360   END
END_PROGRAM

PROGRAM 20TEST
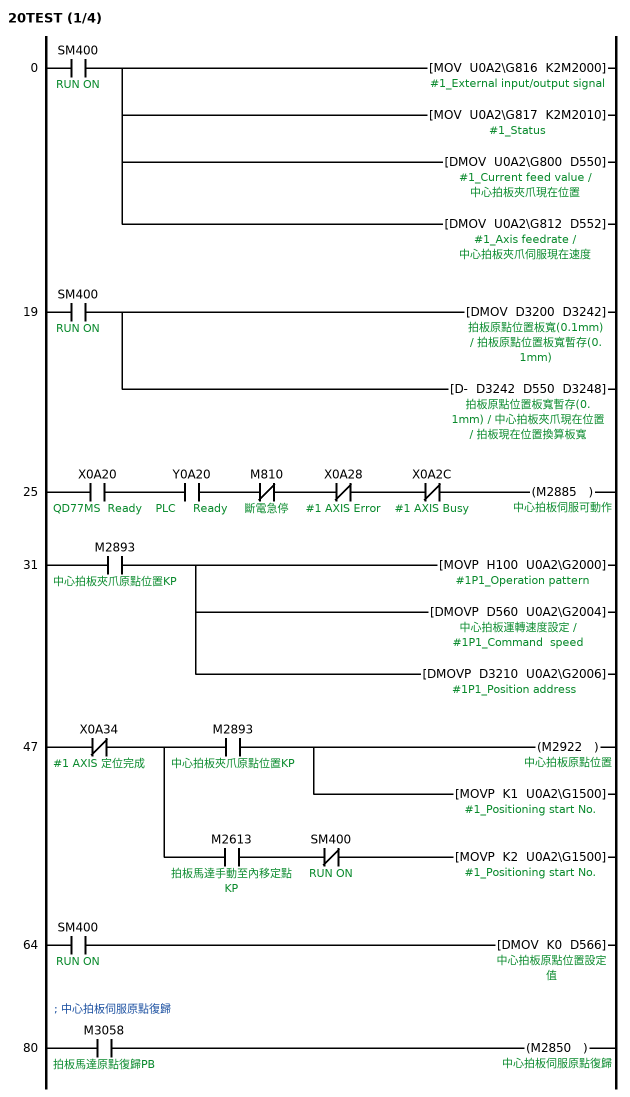
0     LD      SM400  ; RUN ON
      MOV     U0A2\G816 K2M2000  ; #1_External input/output signal / 軸1伺服馬達外極限
      MOV     U0A2\G817 K2M2010  ; #1_Status / Axis01  速度控制
      DMOV    U0A2\G800 D550  ; #1_Current feed value / 中心拍板夾爪現在位置
      DMOV    U0A2\G812 D552  ; #1_Axis feedrate / 中心拍板夾爪伺服現在速度
19    LD      SM400  ; RUN ON
      DMOV    D3200 D3242  ; 拍板原點位置板寬(0.1mm) / 拍板原點位置板寬暫存(0.1mm)
      D-      D3242 D550 D3248  ; 拍板現在位置換算板寬
25    LD      X0A20  ; QD77MS  Ready
      AND     Y0A20  ; PLC     Ready
      ANI     M810  ; 斷電急停
      ANI     X0A28  ; #1 AXIS Error
      ANI     X0A2C  ; #1 AXIS Busy
      OUT     M2885  ; 中心拍板伺服可動作
31    LD      M2893  ; 中心拍板夾爪原點位置KP
      MOVP    H100 U0A2\G2000  ; #1P1_Operation pattern
      DMOVP   D560 U0A2\G2004  ; 中心拍板運轉速度設定 / #1P1_Command  speed
      DMOVP   D3210 U0A2\G2006  ; #1P1_Position address
47    LDI     X0A34  ; #1 AXIS 定位完成
      MPS
      AND     M2893  ; 中心拍板夾爪原點位置KP
      OUT     M2922  ; 中心拍板原點位置
      MOVP    K1 U0A2\G1500  ; #1_Positioning start No.
      MPP
      AND     M2613  ; 拍板馬達手動至內移定點KP
      ANI     SM400  ; RUN ON
      MOVP    K2 U0A2\G1500
64    LD      SM400  ; RUN ON
      DMOV    K0 D566  ; 中心拍板原點位置設定值
; 中心拍板伺服原點復歸
80    LD      M3058  ; 拍板馬達原點復歸PB
      OUT     M2850  ; 中心拍板伺服原點復歸
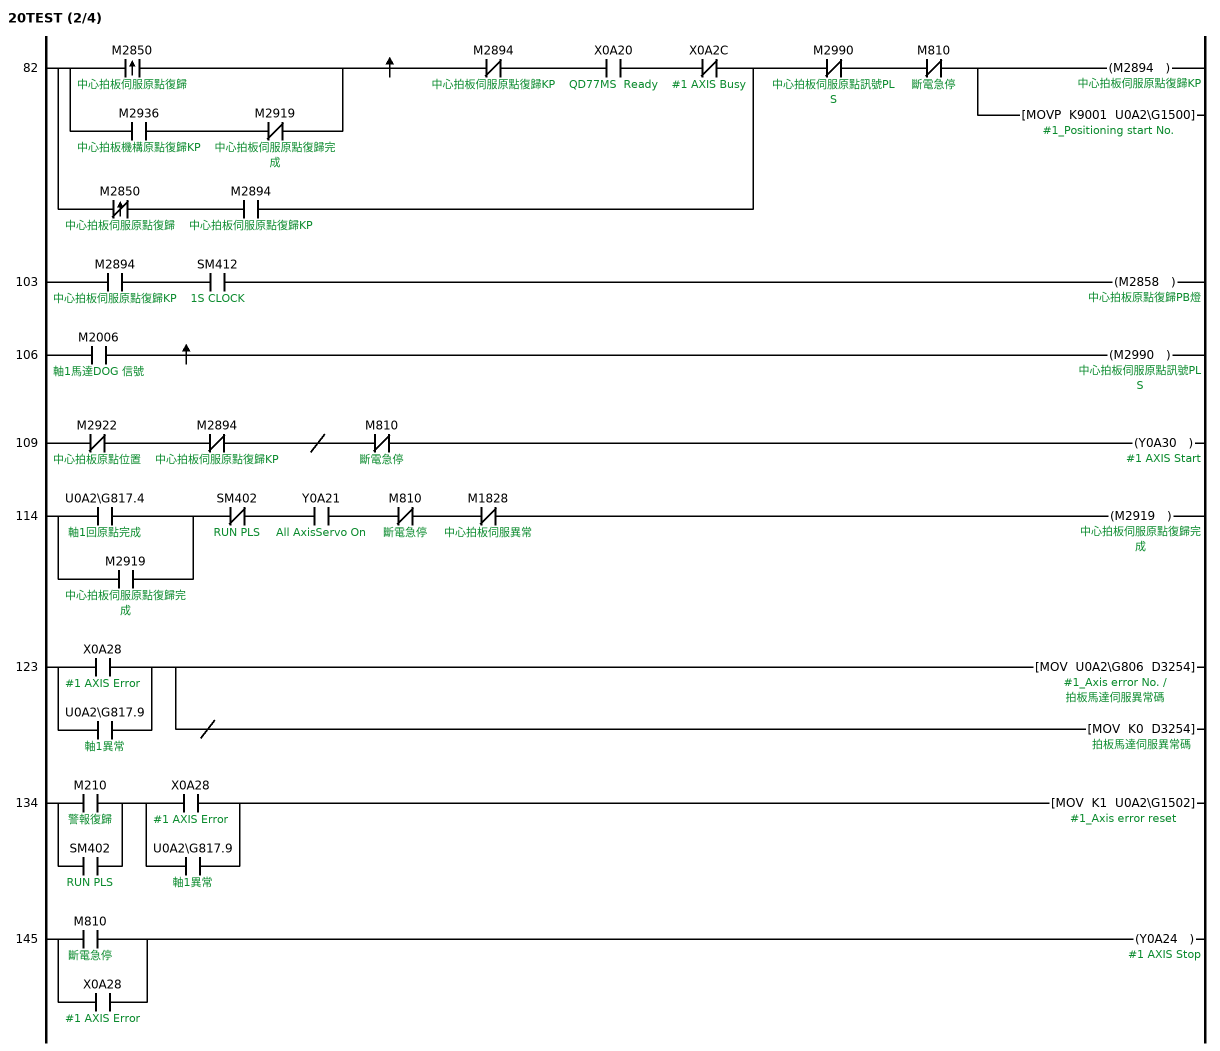
82    LDP     M2850  ; 中心拍板伺服原點復歸
      LD      M2936  ; 中心拍板機構原點復歸KP
      ANI     M2919  ; 中心拍板伺服原點復歸完成
      ORB
      MEP
      ANI     M2894  ; 中心拍板伺服原點復歸KP
      AND     X0A20  ; QD77MS  Ready
      ANI     X0A2C  ; #1 AXIS Busy
      LDPI    M2850  ; 中心拍板伺服原點復歸
      AND     M2894  ; 中心拍板伺服原點復歸KP
      ORB
      ANI     M2990  ; 中心拍板伺服原點訊號PLS
      ANI     M810  ; 斷電急停
      OUT     M2894  ; 中心拍板伺服原點復歸KP
      MOVP    K9001 U0A2\G1500
103   LD      M2894  ; 中心拍板伺服原點復歸KP
      AND     SM412  ; 1S CLOCK
      OUT     M2858  ; 中心拍板原點復歸PB燈
106   LD      M2006  ; 軸1馬達DOG 信號
      MEP
      OUT     M2990  ; 中心拍板伺服原點訊號PLS
109   LDI     M2922  ; 中心拍板原點位置
      ANI     M2894  ; 中心拍板伺服原點復歸KP
      INV
      ANI     M810  ; 斷電急停
      OUT     Y0A30  ; #1 AXIS Start
114   LD      U0A2\G817.4  ; 軸1回原點完成
      OR      M2919  ; 中心拍板伺服原點復歸完成
      ANI     SM402  ; RUN PLS
      AND     Y0A21  ; All AxisServo On
      ANI     M810  ; 斷電急停
      ANI     M1828  ; 中心拍板伺服異常
      OUT     M2919  ; 中心拍板伺服原點復歸完成
123   LD      X0A28  ; #1 AXIS Error
      OR      U0A2\G817.9  ; 軸1異常
      MOV     U0A2\G806 D3254  ; #1_Axis error No. / 拍板馬達伺服異常碼
      INV
      MOV     K0 D3254
134   LD      M210  ; 警報復歸
      OR      SM402  ; RUN PLS
      LD      X0A28  ; #1 AXIS Error
      OR      U0A2\G817.9  ; 軸1異常
      ANB
      MOV     K1 U0A2\G1502  ; #1_Axis error reset
145   LD      M810  ; 斷電急停
      OR      X0A28  ; #1 AXIS Error
      OUT     Y0A24  ; #1 AXIS Stop
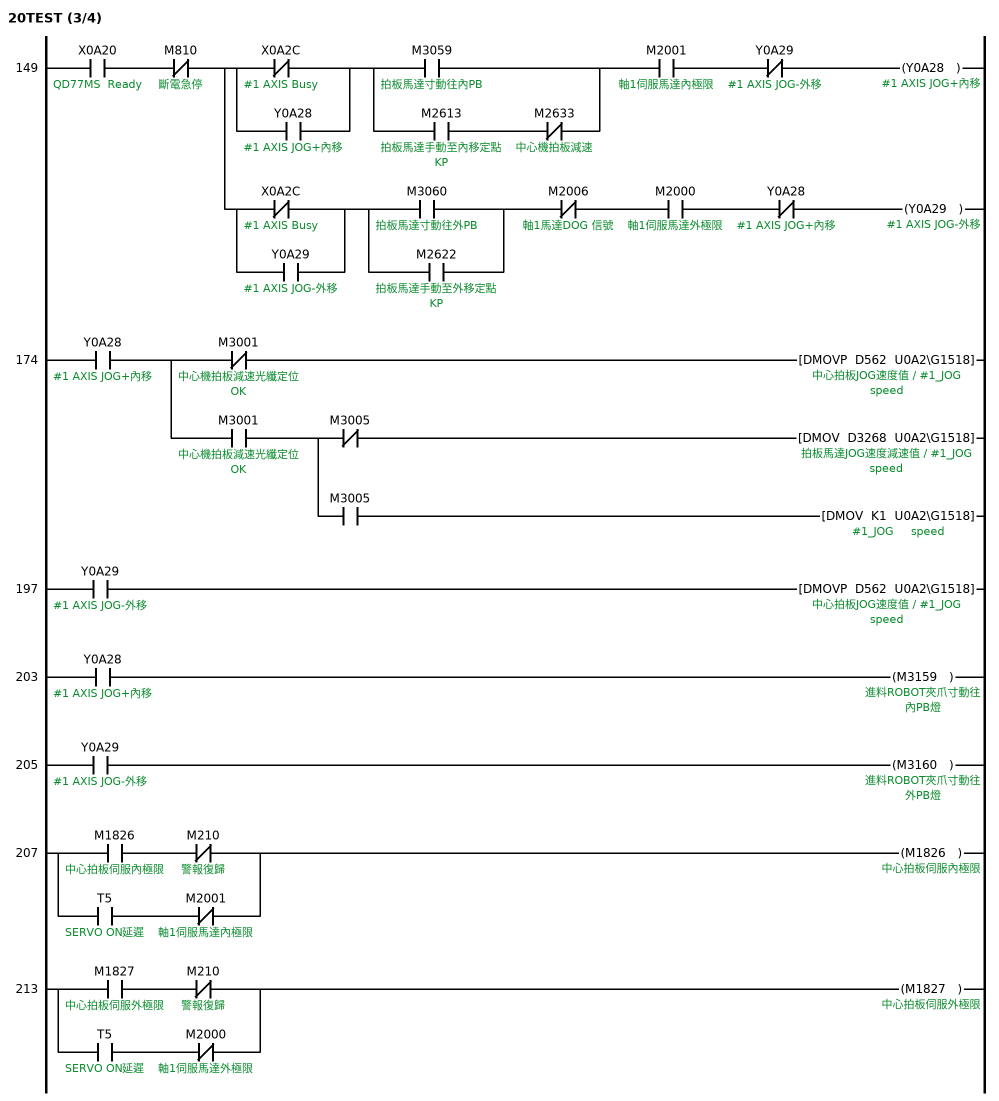
149   LD      X0A20  ; QD77MS  Ready
      ANI     M810  ; 斷電急停
      MPS
      LDI     X0A2C  ; #1 AXIS Busy
      OR      Y0A28  ; #1 AXIS JOG+內移
      ANB
      LD      M3059  ; 拍板馬達寸動往內PB
      LD      M2613  ; 拍板馬達手動至內移定點KP
      ANI     M2633  ; 中心機拍板減速
      ORB
      ANB
      AND     M2001  ; 軸1伺服馬達內極限
      ANI     Y0A29  ; #1 AXIS JOG-外移
      OUT     Y0A28  ; #1 AXIS JOG+內移
      MPP
      LDI     X0A2C  ; #1 AXIS Busy
      OR      Y0A29  ; #1 AXIS JOG-外移
      ANB
      LD      M3060  ; 拍板馬達寸動往外PB
      OR      M2622  ; 拍板馬達手動至外移定點KP
      ANB
      ANI     M2006  ; 軸1馬達DOG 信號
      AND     M2000  ; 軸1伺服馬達外極限
      ANI     Y0A28  ; #1 AXIS JOG+內移
      OUT     Y0A29  ; #1 AXIS JOG-外移
174   LD      Y0A28  ; #1 AXIS JOG+內移
      MPS
      ANI     M3001  ; 中心機拍板減速光纖定位OK
      DMOVP   D562 U0A2\G1518  ; 中心拍板JOG速度值 / #1_JOG     speed
      MPP
      AND     M3001  ; 中心機拍板減速光纖定位OK
      MPS
      ANI     M3005
      DMOV    D3268 U0A2\G1518  ; 拍板馬達JOG速度減速值
      MPP
      AND     M3005
      DMOV    K1 U0A2\G1518
197   LD      Y0A29  ; #1 AXIS JOG-外移
      DMOVP   D562 U0A2\G1518
203   LD      Y0A28  ; #1 AXIS JOG+內移
      OUT     M3159  ; 進料ROBOT夾爪寸動往內PB燈
205   LD      Y0A29  ; #1 AXIS JOG-外移
      OUT     M3160  ; 進料ROBOT夾爪寸動往外PB燈
207   LD      M1826  ; 中心拍板伺服內極限
      ANI     M210  ; 警報復歸
      LD      T5  ; SERVO ON延遲
      ANI     M2001  ; 軸1伺服馬達內極限
      ORB
      OUT     M1826  ; 中心拍板伺服內極限
213   LD      M1827  ; 中心拍板伺服外極限
      ANI     M210  ; 警報復歸
      LD      T5  ; SERVO ON延遲
      ANI     M2000  ; 軸1伺服馬達外極限
      ORB
      OUT     M1827  ; 中心拍板伺服外極限
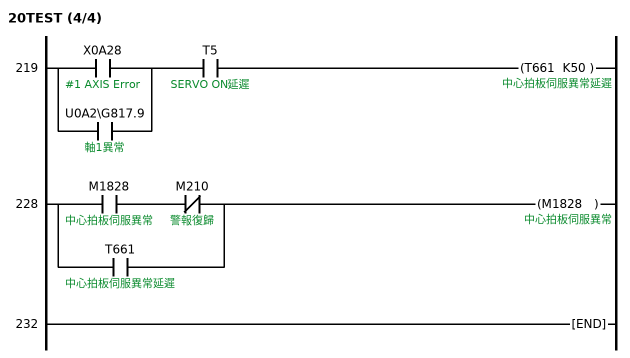
219   LD      X0A28  ; #1 AXIS Error
      OR      U0A2\G817.9  ; 軸1異常
      AND     T5  ; SERVO ON延遲
      OUT     T661 K50  ; 中心拍板伺服異常延遲
228   LD      M1828  ; 中心拍板伺服異常
      ANI     M210  ; 警報復歸
      OR      T661  ; 中心拍板伺服異常延遲
      OUT     M1828  ; 中心拍板伺服異常
232   END
END_PROGRAM

// device comments not shown above
X3D  ; 輸送機輸送馬達  INV41運轉
X31D  ; 30
X327  ; 40
X331  ; 50
X332  ; FR1-DO(31)
X333  ; FR1-DO(32)
X334  ; FR1-DO(33)
X335  ; FR1-DO(34)
X337  ; FR1-DO(36)
X338  ; FR1-DO(37)
X339  ; FR1-DO(38)
X33A  ; FR1-DO(39)
X33B  ; FR1-DO(40)
X33C  ; FR1-DO(41)
X33D  ; FR1-DO(42)
X33E  ; FR1-DO(43)
X33F  ; FR1-DO(44)
X340  ; FR1-DO(45)
X341  ; FR1-DO(46)
X342  ; FR1-DO(47)
X343  ; FR1-DO(48)
X344  ; FR1-DO(49)
X345  ; FR1-DO(50)
X346  ; FR1-DO(51)
X347  ; FR1-DO(52)
X348  ; FR1-DO(53)
X349  ; FR1-DO(54)
X34A  ; FR1-DO(55)
X34B  ; FR1-DO(56)
X34C  ; FR1-DO(57)
X34D  ; FR1-DO(58)
X34E  ; FR1-DO(59)
X34F  ; FR1-DO(60)
X350  ; FR1-DO(61)
X351  ; FR1-DO(62)
X352  ; FR1-DO(63)
X353  ; FR1-DO(64)
X354  ; FR1-DO(65)
X355  ; FR1-DO(66)
X356  ; FR1-DO(67)
X357  ; FR1-DO(68)
X358  ; FR1-DO(69)
X359  ; FR1-DO(70)
X35A  ; FR1-DO(71)
X35B  ; FR1-DO(72)
X35C  ; FR1-DO(73)
X35D  ; FR1-DO(74)
X35E  ; FR1-DO(75)
X35F  ; FR1-DO(76)
X360  ; FR1-DO(77)
X361  ; FR1-DO(78)
X362  ; FR1-DO(79)
X363  ; FR1-DO(80)
X364  ; FR1-DO(81)
X365  ; FR1-DO(82)
X366  ; FR1-DO(83)
X367  ; FR1-DO(84)
X368  ; FR1-DO(85)
X369  ; FR1-DO(86)
X36A  ; FR1-DO(87)
X36B  ; FR1-DO(88)
X36C  ; FR1-DO(89)
X36D  ; FR1-DO(90)
X36E  ; FR1-DO(91)
X36F  ; FR1-DO(92)
X370  ; FR1-DO(93)
X371  ; FR1-DO(94)
X372  ; FR1-DO(95)
X373  ; FR1-DO(96)
X374  ; FR1-DO(97)
X375  ; FR1-DO(98)
X376  ; FR1-DO(99)
X377  ; FR1-DO(100)
X378  ; FR1-DO(101)
X379  ; FR1-DO(102)
X37A  ; FR1-DO(103)
X37B  ; FR1-DO(104)
X37C  ; FR1-DO(105)
X37D  ; FR1-DO(106)
X37E  ; FR1-DO(107)
X37F  ; FR1-DO(108)
X0A03  ; Other station   DataLinkStatus
X0A21  ; Synchronization flag
X0A24  ; #1 AXIS M碼On
X0A25  ; #2 AXIS M碼On
X0A26  ; #3 AXIS M碼On
X0A27  ; #4 AXIS M碼On
X0A2A  ; #3 AXIS Error
X0A2B  ; #4 AXIS Error
X0A2E  ; #3 AXIS Busy
X0A2F  ; #4 AXIS Busy
X0A30  ; #1 AXIS 啟動完成
X0A32  ; #3 AXIS 啟動完成
X0A33  ; #4 AXIS 啟動完成
X0A35  ; #2 AXIS 定位完成
X0A36  ; #3 AXIS 定位完成
X0A37  ; #4 AXIS 定位完成
Y10C  ; @進料連線--取板中
Y31D  ; 30
Y327  ; 40
Y330  ; TR1-DI(31)
Y331  ; TR1-DI(32)-50
Y332  ; TR1-DI(33)
Y333  ; TR1-DI(34)-52
Y334  ; TR1-DI(35)
Y335  ; TR1-DI(36)
Y336  ; TR1-DI(37)-55
Y337  ; TR1-DI(38)
Y338  ; TR1-DI(39)
Y339  ; TR1-DI(40)
Y33A  ; TR1-DI(41)
Y33B  ; TR1-DI(42)
Y33C  ; TR1-DI(43)
Y33D  ; TR1-DI(44)
Y33E  ; TR1-DI(45)
Y33F  ; TR1-DI(46)
Y340  ; TR1-DI(47)
Y341  ; TR1-DI(48)
Y342  ; TR1-DI(49)
Y343  ; TR1-DI(50)
Y344  ; TR1-DI(51)
Y345  ; TR1-DI(52)
Y346  ; TR1-DI(53)
Y347  ; TR1-DI(54)
Y348  ; TR1-DI(55)
Y349  ; TR1-DI(56)
Y34A  ; TR1-DI(57)
Y34B  ; TR1-DI(58)
Y34C  ; TR1-DI(59)
Y34D  ; TR1-DI(60)
Y34E  ; TR1-DI(61)
Y34F  ; TR1-DI(62)
Y350  ; TR1-DI(63)
Y351  ; TR1-DI(64)
Y352  ; TR1-DI(65)
Y353  ; TR1-DI(66)
Y354  ; TR1-DI(67)
Y355  ; TR1-DI(68)
Y356  ; TR1-DI(69)
Y357  ; TR1-DI(70)
Y358  ; TR1-DI(71)
Y359  ; TR1-DI(72)
Y35A  ; TR1-DI(73)
Y35B  ; TR1-DI(74)
Y35C  ; TR1-DI(75)
Y35D  ; TR1-DI(76)
Y35E  ; TR1-DI(77)
Y35F  ; TR1-DI(78)
Y360  ; TR1-DI(79)
Y361  ; TR1-DI(80)
Y362  ; TR1-DI(81)
Y363  ; TR1-DI(82)
Y364  ; TR1-DI(83)
Y365  ; TR1-DI(84)
Y366  ; TR1-DI(85)
Y367  ; TR1-DI(86)
Y368  ; TR1-DI(87)
Y369  ; TR1-DI(88)
Y36A  ; TR1-DI(89)
Y36B  ; TR1-DI(90)
Y36C  ; TR1-DI(91)
Y36D  ; TR1-DI(92)
Y36E  ; TR1-DI(93)
Y36F  ; TR1-DI(94)
Y370  ; TR1-DI(95)
Y371  ; TR1-DI(96)
Y372  ; TR1-DI(97)
Y373  ; TR1-DI(98)
Y374  ; TR1-DI(99)
Y375  ; TR1-DI(100)
Y376  ; TR1-DI(101)
Y377  ; TR1-DI(102)
Y378  ; TR1-DI(103)
Y379  ; TR1-DI(104)
Y37A  ; TR1-DI(105)
Y37B  ; TR1-DI(106)
Y37C  ; TR1-DI(107)
Y37D  ; TR1-DI(108)
Y37E  ; TR1-DI(109)
Y37F  ; TR1-DI(110)
Y0A26  ; #3 AXIS Stop
Y0A27  ; #4 AXIS Stop
Y0A2C  ; #3 AXIS JOG+
Y0A2D  ; #3 AXIS JOG-
Y0A2E  ; #4 AXIS JOG+
Y0A2F  ; #4 AXIS JOG-
Y0A32  ; #3 AXIS Start
Y0A33  ; #4 AXIS Start
Y0A34  ; #1 AXIS 執行禁止
Y0A35  ; #2 AXIS 執行禁止
Y0A36  ; #3 AXIS 執行禁止
Y0A37  ; #4 AXIS 執行禁止
M70  ; 昇降上昇位置教導設定PB
M71  ; 昇降上等待位置教導設定PB
M73  ; 昇降下降位置教導設定PB
M76  ; 下料鼓風機自動
M79  ; 下料鼓風機手動
M190  ; 上料掉板後原點復歸
M191  ; 上料掉板後原點復歸STOP
M237  ; 上料夾爪可伸出KP
M332  ; 進料輸送停止
M333  ; 進料輸送減速KP
M552  ; 進料集塵鼓風機手動運轉
M553  ; 出料集塵鼓風機手動運轉
M554  ; 進出料集塵鼓風機自動運轉
M602  ; #13 風車PB
M603  ; #14 風車PB
M604  ; #15 風車PB
M605  ; #16 風車PB
M606  ; #17 風車PB
M622  ; #13 電熱PB
M623  ; #14 電熱PB
M624  ; #15 電熱PB
M625  ; #16 電熱PB
M626  ; #17 電熱PB
M639  ; 排氣風壓檢知異常警報
M659  ; 排氣風壓檢知異常警報PLS
M732  ; #13 風車訊號
M733  ; #14 風車訊號
M734  ; #15 風車訊號
M735  ; #16 風車訊號
M736  ; #17 風車訊號
M740  ; #01 進氣風車訊號
M741  ; #02 進氣風車訊號
M742  ; #03 進氣風車訊號
M743  ; #04 進氣風車訊號
M744  ; #05 進氣風車訊號
M745  ; #06 進氣風車訊號
M746  ; #07 進氣風車訊號
M747  ; #08 進氣風車訊號
M748  ; #09 進氣風車訊號
M749  ; #10 進氣風車訊號
M750  ; #11 進氣風車訊號
M751  ; #12 進氣風車訊號
M792  ; #13 電熱訊號
M793  ; #14 電熱訊號
M794  ; #15 電熱訊號
M795  ; #16 電熱訊號
M796  ; #17 電熱訊號
M805  ; 上料夾爪短程縮回KP
M832  ; #13 溫度到達KP
M833  ; #14 溫度到達KP
M834  ; #15 溫度到達KP
M835  ; #16 溫度到達KP
M836  ; #17 溫度到達KP
M1304  ; 進料段無板
M1305  ; 進料定位有板
M1426  ; 備用風車啟動PLS
M1427  ; 備用風車啟動PLS
M1526  ; 備用風車停止PLS
M1527  ; 備用風車停止PLS
M2003  ; Axis01  STOP
M2008  ; Axis01  伺服啟動
M2011  ; Axis01  速度轉換位置
M2012  ; Axis01  命令近點
M2013  ; Axis01  歸零要求
M2014  ; Axis01  歸零完成
M2018  ; Axis01  伺服啟動
M2019  ; Axis01  伺服啟動異常
M2020  ; Axis01  移載異常
M2021  ; Axis01  移載警告
M2022  ; Axis01  寸動可運轉
M2023  ; Axis01  命令可運轉
M2024  ; Axis01  歸零完成PLS
M2025  ; Axis01  DO HOME
M2026  ; Axis01  啟動完成
M2027  ; Axis01  DO HOMO 完成
M2028  ; Axis01  要求回原點
M2029  ; Axis01  己回原點
M2030  ; Axis01  移載位置01
M2031  ; Axis01  移載位置02
M2032  ; Axis01  移載位置03
M2033  ; Axis01  移載位置04
M2034  ; Axis01  移載位置05
M2035  ; Axis01  移載位置06
M2036  ; Axis01  移載位置07
M2037  ; Axis01  移載位置08
M2038  ; Axis01  移載位置09
M2039  ; Axis01  移載位置10
M2040  ; Axis01  位置01  訊號
M2041  ; Axis01  位置02  訊號
M2042  ; Axis01  位置03  訊號
M2043  ; Axis01  位置04  訊號
M2044  ; Axis01  位置05  訊號
M2045  ; Axis01  位置06  訊號
M2046  ; Axis01  位置07  訊號
M2047  ; Axis01  位置08  訊號
M2048  ; Axis01  位置09  訊號
M2049  ; Axis01  位置10  訊號
M2050  ; Axis01  READY ON
M2051  ; Axis01  Servo ON
M2054  ; Axis01  Zero point pass
M2055  ; Axis01  In-position
M2056  ; Axis01  Zero speed
M2057  ; Axis01  Torque limit
M2063  ; Axis01  Servo alarm
M2064  ; Axis01  Servo warning
M2070  ; Axis01  速度控制
M2071  ; Axis01  速度轉換位置
M2072  ; Axis01  命令近點
M2073  ; Axis01  歸零要求
M2074  ; Axis01  歸零完成
M2082  ; Axis01  M code ON
M2083  ; Axis01  Error detection
M2084  ; Axis01  Start complete
M2085  ; Axis01  Positioning complete
M2103  ; Axis02  STOP
M2108  ; Axis02  伺服啟動
M2111  ; Axis02  速度轉換位置
M2112  ; Axis02  命令近點
M2113  ; Axis02  歸零要求
M2114  ; Axis02  歸零完成
M2118  ; Axis02  伺服啟動
M2119  ; Axis02  伺服啟動異常
M2120  ; Axis02  移載異常
M2121  ; Axis02  移載警告
M2122  ; Axis02  寸動可運轉
M2123  ; Axis02  命令可運轉
M2124  ; Axis02  歸零完成PLS
M2125  ; Axis02  DO HOME
M2126  ; Axis02  啟動完成
M2127  ; Axis02  DO HOMO 完成
M2128  ; Axis02  要求回原點
M2129  ; Axis02  己回原點
M2130  ; Axis02  移載位置01
M2131  ; Axis02  移載位置02
M2132  ; Axis02  移載位置03
M2133  ; Axis02  移載位置04
M2134  ; Axis02  移載位置05
M2135  ; Axis02  移載位置06
M2136  ; Axis02  移載位置07
M2137  ; Axis02  移載位置08
M2138  ; Axis02  移載位置09
M2139  ; Axis02  移載位置10
M2140  ; Axis02  位置01  訊號
M2141  ; Axis02  位置02  訊號
M2142  ; Axis02  位置03  訊號
M2143  ; Axis02  位置04  訊號
M2144  ; Axis02  位置05  訊號
M2145  ; Axis02  位置06  訊號
M2146  ; Axis02  位置07  訊號
M2147  ; Axis02  位置08  訊號
M2148  ; Axis02  位置09  訊號
M2149  ; Axis02  位置10  訊號
M2150  ; Axis02  READY ON
M2151  ; Axis02  Servo ON
M2154  ; Axis02  Zero point pass
M2155  ; Axis02  In-position
M2156  ; Axis02  Zero speed
M2157  ; Axis02  Torque limit
M2163  ; Axis02  Servo alarm
M2164  ; Axis02  Servo warning
M2170  ; Axis02  速度控制
M2171  ; Axis02  速度轉換位置
M2172  ; Axis02  命令近點
M2173  ; Axis02  歸零要求
M2174  ; Axis02  歸零完成
M2182  ; Axis02  M code ON
M2183  ; Axis02  Error detection
M2184  ; Axis02  Start complete
M2185  ; Axis02  Positioning complete
M2707  ; A6Ini_軟板到位
M2718  ; A6Ini_初始化失敗
M2721  ; A6Auto_檢查有無板
M2722  ; A6Auto_檢查無板
M2723  ; A6Auto_平台下降
M2724  ; A6Auto_前後擋退開
M2725  ; A6Auto_左右擋退開
M2726  ; A6Auto_左右壓板退開
M2727  ; A6Auto_C/V收板請求
M2728  ; A6Auto_C/V收板Busy
M2729  ; A6Auto_C/V收板到位
M2859  ; 中心拍板伺服寸動往內PB燈
M2860  ; 中心拍板伺服寸動往外PB燈
M2890  ; 中心拍板伺服設定位置KP
M2900  ; 中心拍板伺服內極限燈
M2901  ; 中心拍板設定位置燈
M2903  ; 中心拍板夾爪原點位置燈
M2904  ; 中心拍板夾爪伺服原點燈
M2905  ; 中心拍板夾爪伺服外極限燈
M2910  ; 中心拍板設定位置
M2912  ; 中心拍板原點位置
M2920  ; 中心拍板設定位置
M3090  ; 拍板馬達伺服原點訊號PLS1
M3156  ; 拍板馬達至原點PB燈
M3158  ; 拍板馬達原點復歸PB燈
M3188  ; 拍板馬達伺服原點復歸
M3258  ; 拍板馬達伺服原點位置自動
M3319  ; 拍板馬達伺服原點復歸OK
M3358  ; 拍板馬達伺服原點位置手動
M3385  ; 拍板馬達伺服可動作
M3390  ; 拍板馬達設定位置KP
M3393  ; 拍板馬達原點位置KP
M3394  ; 拍板馬達伺服原點復歸KP
M3395  ; 拍板馬達伺服開機原點復歸KP
M3400  ; 拍板馬達伺服內極限燈
M3403  ; 拍板馬達原點位置燈
M3405  ; 拍板馬達伺服外極限燈
M3410  ; 拍板馬達設定位置
M3412  ; 拍板馬達原點位置
M3422  ; 拍板馬達原點位置
M4678  ; 拍板馬達伺服異常
M4704  ; 生產片數到達
M4713  ; 拍板馬達伺服運轉逾時異常
M4716  ; 拍板馬達伺服內極限
M4717  ; 拍板馬達伺服外極限
M4917  ; 刪除配方名稱
M4921  ; 出口計數
M4922  ; 爐內限制異常
M4923  ; 出口計數
M4925  ; 卡板不警報
M4930  ; 點燈運轉KP
M4931  ; 點燈停止
M4932  ; 上位下啟動訊號
M4933  ; PP_SELECT點燈用保持
M4937  ; 上位要儲存配方
M4950  ; 點燈中請稍待指示
M4951  ; 熄點燈冷卻中請稍待指示
M4953  ; 熄燈OK狀態
M4956  ; 輸送機停止熄燈
M4990  ; 密碼ENT
M4992  ; 密碼ENT Keep
M4993  ; 參數設定取消PB
M4994  ; 參數設定取消PLS
M4996  ; 離線測試用
M5034  ; 輸送運轉未加熱完成
M5101  ; 三色紅燈
M5102  ; 三色綠燈
M5215  ; Barcod啟動固定式完成
M5217  ; 門,(1)(2),PPID,配方名稱比對不對
M5314  ; 配方刪除
M5315  ; 配方儲存
M5316  ; 呼叫Q的配方
M5317  ; 比對配方用
M5318  ; 自動
M5319  ; 手動
M5321  ; 自動啟動
M5325  ; 對話視窗關閉
M5326  ; 配方新增
M5327  ; 配方修改
M5328  ; 配方刪除
M5329  ; 機構異常警報
M5347  ; 配方Barcode掃描
M5348  ; 工單輸入
M5349  ; Barcod啟動固定式
M5350  ; Bey Pass PB
M5351  ; 自動PB
M5352  ; 連線開放OP控制
M5353  ; 確認(101頁)人機SET
M5354  ; 確認(102頁)人機SET
M6059  ; Host刪除配方
M6060  ; Host刪除配方完成
M6140  ; 要求上位回讀工單板號右爐
M6141  ; 要求上位回讀工單右爐
M6231  ; 上位要儲存配方
M6300  ; 緊急停止開關異常
M6301  ; 逆相繼電器異常
M6302  ; 入口卡板異常
M6303  ; 出口卡板異常
M6304  ; UV門防止打開開關異常
M6305  ; 上排風風車過載
M6306  ; 下排風風車過載
M6307  ; 安定器冷卻風扇過載
M6308  ; 第一燈溫度異常
M6309  ; 下燈1點燈異常
M6310  ; 下燈2點燈異常
M6311  ; 上燈1點燈異常
M6312  ; 上燈2點燈異常
M6313  ; 變頻機異常
M6314  ; 出料連線異常
M6315  ; 爐內限制數量異常
M6316  ; PLC Low Battery
M6317  ; 進氣冷卻風扇過載
M6318  ; 燈箱冷卻風扇過載
M6319  ; 輸送運轉未點燈警報
M6320  ; 點燈中輸送停止未運轉
M6321  ; 板子有進沒出m231沒滅
M6322  ; 輸送馬達過載異常
M6323  ; 網偏前警報
M6324  ; 網偏後警報
M6325  ; 燈箱冷卻風扇過載
M6326  ; 進氣冷卻風扇過載
M6327  ; 網偏警報熄燈計時
M6328  ; 第二燈溫度異常
M6330  ; UV點燈後30秒不可選擇提示
M6331  ; 下燈1管保養時間到達
M6332  ; 下燈2管保養時間到達
M6333  ; 上燈1管保養時間到達
M6334  ; 上燈2管保養時間到達
M6335  ; 滾輪保養時間到達
M6336  ; 輸送馬達過載異常
M6339  ; 節能省電啟動
M6340  ; 出口卡板異常
M6344  ; 安全門開啟時熄燈選擇    (on熄燈)
M6345  ; 卡板熄燈
M6349  ; 下燈1   點燈失敗
M6350  ; 下燈2   點燈失敗
M6351  ; 上燈1   點燈失敗
M6352  ; 上燈2   點燈失敗
M6607  ; Host刪除配方自保持
M6608  ; Host刪除配方自清除保持
M6610  ; 比對M700~M715都等於零
M6611  ; 比對M716~M731都等於零
M6854  ; 機台再IDEL
M6999  ; 三色綠燈
M7001  ; 三色紅燈
M7999  ; 暫時不開
T8  ; 上料伺服自動復歸次數未到計時
T11  ; 上料伺服自動復歸計時
T12  ; 上料手臂夾爪夾自動延遲
T13  ; 上料昇降伺服運轉延遲
T16  ; 昇降上昇位置教導延遲
T17  ; 昇降上等待位置教導延遲
T19  ; 昇降下降位置教導延遲
T39  ; 下料鼓風機自動停止
T47  ; 進料集塵鼓風機PB延遲
T48  ; 出料集塵鼓風機PB延遲
T49  ; 集塵鼓風機運轉停止延遲
T54  ; 進料段無板延遲
T56  ; ROBOT外部循環啟動計時
T59  ; HMI-LAMP輸送機滾輪輸送OUT運轉OFF
T68  ; 進料輸送減速光電延遲
T112  ; #13 風車PB延遲
T113  ; #14 風車PB延遲
T114  ; #15 風車PB延遲
T115  ; #16 風車PB延遲
T116  ; #17 風車PB延遲
T132  ; #13 電熱PB延遲
T133  ; #14 電熱PB延遲
T134  ; #15 電熱PB延遲
T135  ; #16 電熱PB延遲
T136  ; #17 電熱PB延遲
T139  ; #17 低溫警報
T152  ; #13 低溫警報
T159  ; 進料輸送夾爪夾板異常延遲
T163  ; 進料輸送垂直異常延遲
T164  ; 進料輸送水平異常延遲
T165  ; 上料夾爪長程伸異常延遲
T166  ; 上料夾爪長程縮異常延遲
T188  ; 進料輸送運轉逾時
T190  ; 進料輸送掉板異常延遲
T191  ; 上料夾爪掉板異常延遲
T196  ; 進料空氣壓力異常延時
T200  ; 進料輸送停止時間延遲
T240  ; #01 進氣風車PB延遲
T241  ; #02 進氣風車PB延遲
T242  ; #03 進氣風車PB延遲
T243  ; #04 進氣風車PB延遲
T244  ; #05 進氣風車PB延遲
T245  ; #06 進氣風車PB延遲
T246  ; #07 進氣風車PB延遲
T247  ; #08 進氣風車PB延遲
T248  ; #09 進氣風車PB延遲
T249  ; #10 進氣風車PB延遲
T250  ; #11 進氣風車PB延遲
T251  ; #12 進氣風車PB延遲
T400  ; #01 風車INV運轉計時
T401  ; #02 風車INV運轉計時
T402  ; #03 風車INV運轉計時
T403  ; #04 風車INV運轉計時
T404  ; #05 風車INV運轉計時
T405  ; #06 風車INV運轉計時
T406  ; #07 風車INV運轉計時
T407  ; #08 風車INV運轉計時
T408  ; #09 風車INV運轉計時
T409  ; #10 風車INV運轉計時
T410  ; #11 風車INV運轉計時
T411  ; #12 風車INV運轉計時
T412  ; #13 風車INV運轉計時
T413  ; #14 風車INV運轉計時
T414  ; #15 風車INV運轉計時
T415  ; #16 風車INV運轉計時
T421  ; 出料風車INV運轉計時
T425  ; 進料輸送INV運轉計時
D22  ; 昇降伺服設定參數
D23  ; 昇降伺服異常碼
D24  ; 昇降伺服異常碼
D35  ; 年*10000
D37  ; 月*100
D39  ; 人機時間年月日
D41  ; 進料輸送停止時間延遲
D150  ; 人機參數密碼
D207  ; 取板基準點板長(0.1mm)
D220  ; 上料手臂取板位置換算
D221  ; 上料手臂取板位置暫存
D222  ; 上料手臂取板位置暫存
D249  ; 上料手臂夾爪現在位置換算板寬
D251  ; 上料手臂夾爪現在位置
D253  ; 上料手臂夾爪伺服現在速度
D261  ; 上料手臂夾爪運轉速度設定
D263  ; 上料手臂夾爪JOG速度值
D265  ; 上料手臂夾爪設定位置設定值
D267  ; 上料手臂夾爪原點位置設定值
D297  ; 總生產量Hi
D301  ; 本班產量履歷2
D302  ; 本班產量履歷3
D303  ; 本班產量履歷4
D304  ; 本班產量履歷5
D305  ; 本班產量履歷6
D306  ; 本班產量履歷7
D307  ; 本班產量履歷8
D308  ; 本班產量履歷9
D309  ; 本班產量履歷10
D310  ; 本班產量履歷11
D311  ; 本班產量履歷12
D312  ; 本班產量履歷13
D313  ; 本班產量履歷14
D314  ; 本班產量履歷15
D315  ; 本班產量履歷16
D316  ; 本班產量履歷17
D317  ; 本班產量履歷18
D318  ; 本班產量履歷19
D319  ; 本班產量履歷20
D320  ; 本班產量履歷21
D321  ; 本班產量履歷22
D322  ; 本班產量履歷23
D323  ; 本班產量履歷24
D324  ; 本班產量履歷25
D331  ; 現在時間時分2
D332  ; 現在時間時分3
D333  ; 現在時間時分4
D334  ; 現在時間時分5
D335  ; 現在時間時分6
D336  ; 現在時間時分7
D337  ; 現在時間時分8
D338  ; 現在時間時分9
D339  ; 現在時間時分10
D340  ; 現在時間時分11
D341  ; 現在時間時分12
D342  ; 現在時間時分13
D343  ; 現在時間時分14
D344  ; 現在時間時分15
D345  ; 現在時間時分16
D346  ; 現在時間時分17
D347  ; 現在時間時分18
D348  ; 現在時間時分19
D349  ; 現在時間時分20
D350  ; 現在時間時分21
D351  ; 現在時間時分22
D352  ; 現在時間時分23
D353  ; 現在時間時分24
D354  ; 現在時間時分25
D395  ; 月保養時間現在值
D397  ; 季保養時間現在值
D399  ; 年保養時間現在值
D400  ; PLC=>SV1
D401  ; PLC=>SV2
D402  ; PLC=>SV3
D403  ; PLC=>SV4
D404  ; PLC=>SV5
D405  ; PLC=>SV6
D406  ; PLC=>SV7
D407  ; PLC=>SV8
D408  ; PLC=>SV9
D409  ; PLC=>SV10
D420  ; PV1=>PLC
D421  ; PV2=>PLC
D422  ; PV3=>PLC
D423  ; PV4=>PLC
D424  ; PV5=>PLC
D425  ; PV6=>PLC
D426  ; PV7=>PLC
D427  ; PV8=>PLC
D428  ; PV9=>PLC
D429  ; PV10=>PLC
D440  ; SV1=>PLC
D441  ; SV2=>PLC
D442  ; SV3=>PLC
D443  ; SV4=>PLC
D444  ; SV5=>PLC
D445  ; SV6=>PLC
D446  ; SV7=>PLC
D447  ; SV8=>PLC
D448  ; SV9=>PLC
D449  ; SV10=>PLC
D548  ; 中心拍板現在位置換算板寬
D549  ; 中心拍板現在位置換算板寬
D551  ; 中心拍板夾爪現在位置
D553  ; 中心拍板夾爪伺服現在速度
D554  ; 中心拍板伺服異常碼
D561  ; 中心拍板運轉速度設定
D563  ; 中心拍板JOG速度值
D564  ; 中心拍板設定位置設定值
D565  ; 中心拍板設定位置設定值
D567  ; 中心拍板原點位置設定值
D641  ; 烘烤時間SEC
D701  ; 月保養時數
D711  ; 季保養時數
D721  ; 年保養時數
D809  ; 排氣風壓檢知異常警報
D859  ; 排氣風壓檢知異常警報暫存
D1001  ; 系統時間年月日00
D1002  ; 系統時間年月日01
D1003  ; 系統時間年月日01
D1004  ; 系統時間年月日02
D1005  ; 系統時間年月日02
D1006  ; 系統時間年月日03
D1007  ; 系統時間年月日03
D1008  ; 系統時間年月日04
D1009  ; 系統時間年月日04
D1010  ; 系統時間年月日05
D1011  ; 系統時間年月日05
D1012  ; 系統時間年月日06
D1013  ; 系統時間年月日06
D1014  ; 系統時間年月日07
D1015  ; 系統時間年月日07
D1016  ; 系統時間年月日08
D1017  ; 系統時間年月日08
D1018  ; 系統時間年月日09
D1019  ; 系統時間年月日09
D1020  ; 系統時間年月日10
D1021  ; 系統時間年月日10
D1022  ; 系統時間年月日11
D1023  ; 系統時間年月日11
D1024  ; 系統時間年月日12
D1025  ; 系統時間年月日12
D1026  ; 系統時間年月日13
D1027  ; 系統時間年月日13
D1028  ; 系統時間年月日14
D1029  ; 系統時間年月日14
D1030  ; 系統時間年月日15
D1031  ; 系統時間年月日15
D1032  ; 系統時間年月日16
D1033  ; 系統時間年月日16
D1034  ; 系統時間年月日17
D1035  ; 系統時間年月日17
D1036  ; 系統時間年月日18
D1037  ; 系統時間年月日18
D1038  ; 系統時間年月日19
D1039  ; 系統時間年月日19
D1040  ; 系統時間年月日20
D1041  ; 系統時間年月日20
D1042  ; 系統時間年月日21
D1043  ; 系統時間年月日21
D1044  ; 系統時間年月日22
D1045  ; 系統時間年月日22
D1046  ; 系統時間年月日23
D1047  ; 系統時間年月日23
D1048  ; 系統時間年月日24
D1049  ; 系統時間年月日24
D2000  ; TR1 ROBOT取板點(補償)X
D2001  ; TR1 ROBOT取板點(補償)Y
D2002  ; TR1 ROBOT取板點(補償)Z
D2008  ; TR1 ROBOT放板點(補償)X
D2009  ; TR1 ROBOT放板點(補償)Y
D2010  ; TR1 ROBOT放板點(補償)Z
D2101  ; TR1(R31)手臂取板點(補償)X
D2102  ; TR1(R32)手臂取板點(補償)Y
D2103  ; TR1(R33)手臂取板點(補償)Z
D2104  ; TR1(R34)手臂取板點(補償)角度
D2105  ; TR1(R35)手臂放板點(補償)X
D2106  ; TR1(R36)手臂放板點(補償)Y
D2107  ; TR1(R37)手臂放板點(補償)Z
D2109  ; TR1(R39)板長尺寸偏差量(0.1mm)
D2110  ; TR1(R40)
D2111  ; TR1(R41)
D2112  ; TR1(R42)
D2113  ; TR1(R43)
D2114  ; TR1(R44)
D2115  ; TR1(R45)
D2502  ; 人機手臂取板點(補償)Y
D2503  ; 人機手臂取板點(補償)Z
D2505  ; 人機手臂放板點(補償)Y
D2506  ; 人機手臂放板點(補償)Z
D2509  ; 板長尺寸偏差量計算(0.1mm)
D3243  ; 拍板原點位置板寬暫存(0.1mm)
D3250  ; 拍板馬達現在位置
D3252  ; 拍板馬達現在速度
D3260  ; 拍板馬達運轉速度設定
D3262  ; 拍板馬達JOG速度值
D3266  ; 拍板馬達原點位置設定值
D3302  ; 當前使用配方RecipeID#04/03
D3303  ; 當前使用配方RecipeID#06/05
D3304  ; 當前使用配方RecipeID#08/07
D3305  ; 當前使用配方RecipeID#10/09
D3306  ; 當前使用配方RecipeID#12/11
D3307  ; 當前使用配方RecipeID#14/13
D3308  ; 當前使用配方RecipeID#16/15
D3309  ; 當前使用配方RecipeID#18/17
D3310  ; 當前使用配方RecipeID#20/19
D3311  ; 當前使用配方RecipeID#22/21
D3312  ; 當前使用配方RecipeID#24/23
D3313  ; 當前使用配方RecipeID#26/25
D3314  ; 當前使用配方RecipeID#28/27
D3315  ; 當前使用配方RecipeID#30/29
D3316  ; 當前使用配方RecipeID#32/31
D3317  ; 當前使用配方RecipeID#34/33
D3318  ; 當前使用配方RecipeID#36/35
D3319  ; 當前使用配方RecipeID#38/37
D3320  ; 當前使用配方RecipeID#40/39
D3322  ; 當前使用配方第02槽電熱設定
D3323  ; 當前使用配方第03槽電熱設定
D3324  ; 當前使用配方第04槽電熱設定
D3325  ; 當前使用配方第05槽電熱設定
D3326  ; 當前使用配方第06槽電熱設定
D3327  ; 當前使用配方第07槽電熱設定
D3328  ; 當前使用配方第08槽電熱設定
D3329  ; 當前使用配方第09槽電熱設定
D3330  ; 當前使用配方第10槽電熱設定
D3331  ; 當前使用配方第11槽電熱設定
D3332  ; 當前使用配方第12槽電熱設定
D3390  ; HMI-編輯RecipeID#22/21
D3391  ; HMI-編輯RecipeID#24/23
D3392  ; HMI-編輯RecipeID#26/25
D3393  ; HMI-編輯RecipeID#28/27
D3394  ; HMI-編輯RecipeID#30/29
D3395  ; HMI-編輯RecipeID#32/31
D3396  ; HMI-編輯RecipeID#34/33
D3397  ; HMI-編輯RecipeID#36/35
D3398  ; HMI-編輯RecipeID#38/37
D3399  ; HMI-編輯RecipeID#40/39
D3420  ; HMI-編輯爐內烘烤時間計算-2(秒)
D3422  ; HMI-編輯爐內烘烤時間計算-2(分)
D4940  ; SP.SOC OPEN指令控制數據
D4944  ; SP.SOC SND指令結束元件
D4950  ; SP.SOC  SND指令控制數據
D4952  ; SP.SOC  RCV指令控制數據
D4954  ; SP.SOC  CLOSE指令控制數據
D5105  ; ATMA->GP板長mm
D5106  ; ATMA->GP板寬mm
D5508  ; [ED-02] 配方異動型態
D5514  ; 配方組別計算-2-(1)
D10070  ; 比對START字串
D10071  ; 比對STOP字串
D10072  ; 比對PP_SELECT字串
D10074  ; 比對配方名稱為零可儲存位址
D10076  ; 名稱有一樣的是更新=50要新增
D10077  ; 比對PAUSE字串
D10078  ; 比對RESUME字串
D10081  ; 上位下配方比對結果
D10083  ; 上位下的組別右門(比對出來的)
D10084  ; 名稱GO-LOCAL比對結果
D10085  ; 名稱PPID比對結果
D10086  ; 上位下配方比對結果
D10087  ; 上位下的組別左門(比對出來的)
D10661  ; SECS_上位下PAUSE指令
D10662  ; SECS_上位下PAUSE指令
D13531  ; 第01槽電熱實際溫度PV(FLT)
D13533  ; 第02槽電熱實際溫度PV(FLT)
D13535  ; 第03槽電熱實際溫度PV(FLT)
D13537  ; 第04槽電熱實際溫度PV(FLT)
D13539  ; 第05槽電熱實際溫度PV(FLT)
D13541  ; 第06槽電熱實際溫度PV(FLT)
D13543  ; 第07槽電熱實際溫度PV(FLT)
D13545  ; 第08槽電熱實際溫度PV(FLT)
D13547  ; 第09槽電熱實際溫度PV(FLT)
D13549  ; 第10槽電熱實際溫度PV(FLT)
D13551  ; 第11槽電熱實際溫度PV(FLT)
D13553  ; 第12槽電熱實際溫度PV(FLT)
D13555  ; 第01槽風壓檢知PV(FLT)
D13557  ; 第02槽風壓檢知PV(FLT)
D13559  ; 第03槽風壓檢知PV(FLT)
D13561  ; 第04槽風壓檢知PV(FLT)
D13563  ; 第05槽風壓檢知PV(FLT)
D13565  ; 第06槽風壓檢知PV(FLT)
D13567  ; 第07槽風壓檢知PV(FLT)
D13569  ; 第08槽風壓檢知PV(FLT)
D13571  ; 第09槽風壓檢知PV(FLT)
D13573  ; 第10槽風壓檢知PV(FLT)
D13575  ; 第11槽風壓檢知PV(FLT)
D13577  ; 第12槽風壓檢知PV(FLT)
L9  ; 爐內掉板不使用PB&LAMP
L3804  ; 第05站  CC-LINK 異常
L3805  ; 第06站  CC-LINK 異常
L3806  ; 第07站  CC-LINK 異常
L3807  ; 第08站  CC-LINK 異常
L3808  ; 第09站  CC-LINK 異常
L3809  ; 第10站  CC-LINK 異常
L3810  ; 第11站  CC-LINK 異常
L3811  ; 第12站  CC-LINK 異常
L3812  ; 第13站  CC-LINK 異常
L3813  ; 第14站  CC-LINK 異常
L3814  ; 第15站  CC-LINK 異常
L3815  ; 第16站  CC-LINK 異常
R1000  ; PASSWORELEVEL 01
R1001  ; PASSWORELEVEL 01
R1002  ; PASSWORELEVEL 02
R1003  ; PASSWORELEVEL 02
R1004  ; PASSWORELEVEL 03
R1005  ; PASSWORELEVEL 03
R1006  ; PASSWORELEVEL 04
R1007  ; PASSWORELEVEL 04
R1008  ; PASSWORELEVEL 05
R1009  ; PASSWORELEVEL 05
R1010  ; PASSWORELEVEL 06
R1011  ; PASSWORELEVEL 06
R1012  ; PASSWORELEVEL 07
R1013  ; PASSWORELEVEL 07
R1014  ; PASSWORELEVEL 08
R1015  ; PASSWORELEVEL 08
R1016  ; PASSWORELEVEL 09
R1017  ; PASSWORELEVEL 09
R1018  ; PASSWORELEVEL 10
R1019  ; PASSWORELEVEL 10
R1020  ; PASSWORELEVEL 11
R1021  ; PASSWORELEVEL 11
R1022  ; PASSWORELEVEL 12
R1023  ; PASSWORELEVEL 12
R1024  ; PASSWORELEVEL 13
R1025  ; PASSWORELEVEL 13
R1026  ; PASSWORELEVEL 14
R1027  ; PASSWORELEVEL 14
R1028  ; PASSWORELEVEL 15
R1029  ; PASSWORELEVEL 15
R5009  ; Default Communication State:Enab
R5010  ; Default Control:ON-LINE/OFF-LINE
R5011  ; Default ON-LINE fail Substate:
R5015  ; Over Write Spool:Enable/Disable
R5018  ; Config Spool:Enable/Disable
R6000  ; 板架計數
ZR0  ; [ED-02] Modify Type
ZR1  ; [ED-02] RecipeID#02/01
ZR2  ; [ED-02] RecipeID#04/03
ZR3  ; [ED-02] RecipeID#06/05
ZR4  ; [ED-02] RecipeID#08/07
ZR5  ; [ED-02] RecipeID#10/09
ZR6  ; [ED-02] RecipeID#12/11
ZR7  ; [ED-02] RecipeID#14/13
ZR8  ; [ED-02] RecipeID#16/15
ZR9  ; [ED-02] RecipeID#18/17
ZR10  ; [ED-02] RecipeID#20/19
ZR11  ; [ED-02] RecipeID#22/21
ZR12  ; [ED-02] RecipeID#24/23
ZR13  ; [ED-02] RecipeID#26/25
ZR14  ; [ED-02] RecipeID#28/27
ZR15  ; [ED-02] RecipeID#30/29
ZR21  ; [ED-02] HEAT-SV #01
ZR22  ; [ED-02] HEAT-SV #02
ZR23  ; [ED-02] HEAT-SV #03
ZR24  ; [ED-02] HEAT-SV #04
ZR25  ; [ED-02] HEAT-SV #05
ZR26  ; [ED-02] HEAT-SV #06
ZR27  ; [ED-02] HEAT-SV #07
ZR28  ; [ED-02] HEAT-SV #08
ZR29  ; [ED-02] HEAT-SV #09
ZR30  ; [ED-02] HEAT-SV #10
ZR31  ; [ED-02] HEAT-SV #11
ZR32  ; [ED-02] HEAT-SV #12
ZR146  ; 上報軟體編號SoftRev
ZR147  ; 上報軟體編號SoftRev
ZR151  ; Code-S7-F23-F25
ZR157  ; 上報儲存配方處理0=OK,3=沒空間
ZR2035  ; SECS_上位下載配方Recipe NO.
ZR2036  ; SECS_上位下載配方RecipeID#02/01
ZR2037  ; SECS_上位下載配方RecipeID#04/03
ZR2038  ; SECS_上位下載配方RecipeID#06/05
ZR2039  ; SECS_上位下載配方RecipeID#08/07
ZR2040  ; SECS_上位下載配方RecipeID#10/09
ZR2041  ; SECS_上位下載配方RecipeID#12/11
ZR2042  ; SECS_上位下載配方RecipeID#14/13
ZR2043  ; SECS_上位下載配方RecipeID#16/15
ZR2044  ; SECS_上位下載配方RecipeID#18/17
ZR2045  ; SECS_上位下載配方RecipeID#20/19
ZR2046  ; SECS_上位下載配方第01槽電熱設定
ZR2047  ; SECS_上位下載配方第02槽電熱設定
ZR2048  ; SECS_上位下載配方第03槽電熱設定
ZR2049  ; SECS_上位下載配方第04槽電熱設定
ZR2050  ; SECS_上位下載配方第05槽電熱設定
ZR2051  ; SECS_上位下載配方第06槽電熱設定
ZR2052  ; SECS_上位下載配方第07槽電熱設定
ZR2053  ; SECS_上位下載配方第08槽電熱設定
ZR2054  ; SECS_上位下載配方第09槽電熱設定
ZR2055  ; SECS_上位下載配方第10槽電熱設定
ZR2056  ; SECS_上位下載配方第11槽電熱設定
ZR2057  ; SECS_上位下載配方第12槽電熱設定
ZR2058  ; SECS_上位下載配方進料步進間隔次
ZR2059  ; SECS_上位下載配方烘烤步進時間設
ZR2060  ; SECS_上位下載配方板材尺寸寬度設
ZR5201  ; SECS_上位配方NO.01
ZR5299  ; SECS_上位配方NO.50
ZR10001  ; 異動暫存RecipeID#02/01
ZR10002  ; 異動暫存RecipeID#04/03
ZR10003  ; 異動暫存RecipeID#06/05
ZR10004  ; 異動暫存RecipeID#08/07
ZR10005  ; 異動暫存RecipeID#10/09
ZR10006  ; 異動暫存RecipeID#12/11
ZR10007  ; 異動暫存RecipeID#14/13
ZR10008  ; 異動暫存RecipeID#16/15
ZR10009  ; 異動暫存RecipeID#18/17
ZR10010  ; 異動暫存RecipeID#20/19
ZR10011  ; 異動暫存RecipeID#22/21
ZR10012  ; 異動暫存RecipeID#24/23
ZR10013  ; 異動暫存RecipeID#26/25
ZR10014  ; 異動暫存RecipeID#28/27
ZR10015  ; 異動暫存RecipeID#30/29
ZR10016  ; 異動暫存RecipeID#32/31
ZR10017  ; 異動暫存RecipeID#34/33
ZR10018  ; 異動暫存RecipeID#36/35
ZR10019  ; 異動暫存RecipeID#38/37
ZR10020  ; 異動暫存RecipeID#40/39
ZR10021  ; 異動暫存第01槽電熱設定
ZR10022  ; 異動暫存第02槽電熱設定
ZR10023  ; 異動暫存第03槽電熱設定
ZR10024  ; 異動暫存第04槽電熱設定
ZR10025  ; 異動暫存第05槽電熱設定
ZR10026  ; 異動暫存第06槽電熱設定
ZR10027  ; 異動暫存第07槽電熱設定
ZR10028  ; 異動暫存第08槽電熱設定
ZR10029  ; 異動暫存第09槽電熱設定
ZR10030  ; 異動暫存第10槽電熱設定
ZR10031  ; 異動暫存第11槽電熱設定
ZR10032  ; 異動暫存第12槽電熱設定
ZR10033  ; 異動暫存進料步進間隔次數設定
ZR10034  ; 異動暫存烘烤步進時間設定
ZR10035  ; 異動暫存板材尺寸寬度設定
ZR10039  ; 異動暫存烘烤時間(分)
P0  ; 初始設定
P5  ; 功能選擇
P10  ; FX2N-2AD
P20  ; FX2N-1PG(昇降)
P90  ; 原點訊號
P100  ; 進料機構
P105  ; 上料機構
P110  ; 下料機構
P120  ; 下料位移機構
P130  ; 電熱啟動停止
P140  ; 風車電熱訊號
P150  ; 產能履歷
P160  ; 設備運轉保養時間
P170  ; 電熱風車異常訊號
P180  ; 一般異常
P190  ; 烘烤時間
D5002.0  ; GP->ATMA_ROBOT準備取板
D5002.1  ; GP->ATMA_ROBOT動作完成
D5102.8  ; ATMA->GP_印刷機連線
D5102.9  ; ATMA->GP_印刷機取板要求
D5102.A  ; ATMA->GP_印刷機動作異常
